# B&R Automation Studio project DuctLines (part 9)

### Program Logical/Uncoiler_1 (IEC)

#### Cyclic.ld
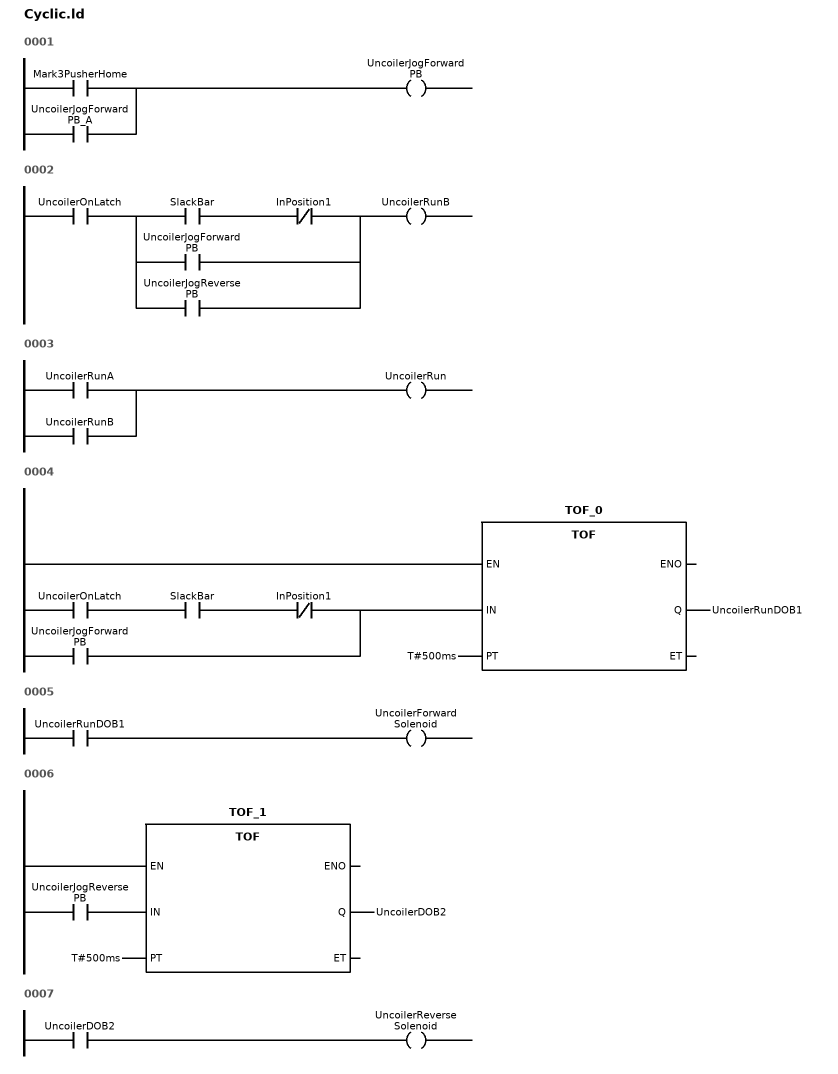
Ladder, written as Structured Text:
```iecst
PROGRAM _CYCLIC
(* Network 1 *)
UncoilerJogForwardPB := Mark3PusherHome OR UncoilerJogForwardPB_A;

(* Network 2 *)
UncoilerRunB := UncoilerOnLatch AND ((SlackBar AND NOT InPosition1) OR UncoilerJogForwardPB OR UncoilerJogReversePB);

(* Network 3 *)
UncoilerRun := UncoilerRunA OR UncoilerRunB;

(* Network 4 *)
TOF_0(IN := (UncoilerOnLatch AND SlackBar AND NOT InPosition1) OR UncoilerJogForwardPB, PT := T#500ms);
UncoilerRunDOB1 := TOF_0.Q;

(* Network 5 *)
UncoilerForwardSolenoid := UncoilerRunDOB1;

(* Network 6 *)
TOF_1(IN := UncoilerJogReversePB, PT := T#500ms);
UncoilerDOB2 := TOF_1.Q;

(* Network 7 *)
UncoilerReverseSolenoid := UncoilerDOB2;
END_PROGRAM
```

### Program Logical/E2Feeder (IEC) - 3/11/19 Punchmaster logic was redundant. Deleted rungs 169-189.

#### Variables.var
```iecst
VAR
	AutoSignal : BOOL;
	BatchCancelUnlatch : BOOL;
	BeadRollFires : BOOL;
	BeadRollUsedUp : BOOL;
	Block_1 : BOOL;
	BrakeLatch : BOOL;
	ButtonBack7 : BOOL;
	ButtonFires : BOOL;
	ButtonUsedUp : BOOL;
	CenterHoleFires : BOOL;
	CenterHoleTime : TIME;
	CenterHoleUsedUp : BOOL;
	CenterPosA : BOOL;
	CenterShuttleIndex : INT;
	ChangeCShuttle : BOOL;
	ChangeJob1 : BOOL;
	ChangeRShuttle : BOOL;
	ClearEncoderSignal : BOOL;
	CleatFires : BOOL;
	CleatUsedUp : BOOL;
	CLPUnlatch : BOOL;
	CoilPowerTripPulse : BOOL;
	CShuttleUnlatch : BOOL;
	CustomLTFires : BOOL;
	CustomLTTime : TIME;
	CustomLTUsedUp : BOOL;
	CustomLTValve : BOOL;
	CustomVFires : BOOL;
	CustomVTime : TIME;
	CustomVUsedUp : BOOL;
	DamperLatch : BOOL;
	DamperResult : DINT;
	DataUpdated : BOOL;
	DDDoneTimer : TON;
	DieDelayDone : BOOL;
	DieUpTime : TIME;
	DirectionDelayDone : BOOL;
	DuctoAutoUnlatch : BOOL;
	FFCLatch : BOOL;
	FiveFootCoil : BOOL;
	FourFootCoil : BOOL;
	FourResult : DINT;
	GapPulse : BOOL;
	GapTP : BOOL;
	GTime : TIME;
	HalfUpdated1 : BOOL;
	HalfUpdated2 : BOOL;
	HolePunchSelecedtSolenoid : BOOL;
	IncPartsMade : BOOL;
	InitMoveSignal : BOOL;
	InPositionBand : REAL := 0.01;
	JobChanging : BOOL;
	JobsDifferent : BOOL;
	LeftHoleFires : BOOL;
	LeftHoleTime : TIME;
	LeftHoleUsedUp : BOOL;
	LeftPosA : BOOL;
	LTFires : BOOL;
	LTTime : TIME;
	LTUsedUp : BOOL;
	MarkAccumulator : REAL;
	MetalEncoderLatch : DINT;
	NewRunJobOk : BOOL;
	NextMoveComplete : BOOL;
	NextMoveLookAgain : BOOL;
	NoShearHits : BOOL;
	OGLatch : BOOL;
	OGResult : DINT;
	OneResult : DINT;
	OutsideLatch : BOOL;
	PartCutOff : BOOL;
	PartRefOK : BOOL;
	PunchCurrentSelect : DINT;
	ReturnCalculated : BOOL;
	ReturnComplete : BOOL;
	ReturnTarget : DINT;
	RightHoleFires : BOOL;
	RightHoleTime : TIME;
	RightHoleUsedUp : BOOL;
	RightPosA : BOOL;
	RollEnableUnlatch : BOOL;
	RShuttleUnlatch : BOOL;
	RTotalInches : REAL;
	RunSpeedCalculated : BOOL;
	SetConnectorChange : BOOL;
	ShearBrakeFires : BOOL;
	ShearBrakeUsedUp : BOOL;
	ShearFires : BOOL;
	ShearHitsLTZero : BOOL;
	shearTime : TIME;
	ShearUsedUp : BOOL;
	SHLT0 : BOOL;
	SixFootCoil : BOOL;
	SmallResult : REAL;
	Step04A : BOOL;
	Step05A : BOOL;
	Step05B : BOOL;
	Step06 : BOOL;
	Step07 : BOOL;
	Step08 : BOOL;
	Step09 : BOOL;
	Step10 : BOOL;
	Step15 : BOOL;
	Step16 : BOOL;
	Step17 : BOOL;
	Step18A : BOOL;
	Step20 : BOOL;
	Step22 : BOOL;
	ThirdOff1 : BOOL;
	ThirdOff2 : BOOL;
	ThirdOff3 : BOOL;
	TON_0 : TON;
	TON_1 : TON;
	TON_10 : TON;
	TON_Warning : TON;
	TP_0 : TP;
	TP_1 : TP;
	TP_2 : TP;
	TP_3 : TP;
	TP_4 : TP;
	TP_5 : TP;
	TP_6 : TP;
	TP_7 : TP;
	TP_8 : TP;
	TP_9 : TP;
	TP_10 : TP;
	UnlatchBender : BOOL;
	UnlatchButtons : BOOL;
	VFires : BOOL;
	VTime : TIME;
	VUsedUp : BOOL;
	Wait1Ready : BOOL;
	Wait2Ready : BOOL;
	Wait3Ready : BOOL;
	WaitCon1 : BOOL;
	WaitCon2 : BOOL;
	ZCOLT0 : BOOL;
	ZCReverseComplete : BOOL;
	ZCSCTimer : TON;
	ZCSettleComplete : BOOL;
	ZeroCropDifference : DINT;
	ZRCTon : TON;
	FinalScan : BOOL;
	ShearAndDieFires : BOOL;
	DieDoneTimer : BOOL;
	TP_11 : TP;
END_VAR
```

#### Action.st
```iecst
ACTION myAction:
	IF ShearHits < 120000 THEN
		ShearHits := ShearHits + 1;
	END_IF;

END_ACTION

ACTION getNextMove:
	(*Find smallest move*)
	(*The shear will always be used*)
	IF getNextMove.x AND NOT getNextMove._x THEN
		FinalScan := TRUE;
	ELSE
		NextMoveDone := TRUE;
		SmallResult := ShearMove;
		IF LTNotchMove < SmallResult AND LTNotchMove > InvalidDistREAL THEN
			SmallResult := LTNotchMove;
		END_IF;
		IF VNotchMove < SmallResult AND VNotchMove > InvalidDistREAL THEN
			SmallResult := VNotchMove;
		END_IF;
		IF LeftHoleMove < SmallResult AND LeftHoleMove > InvalidDistREAL THEN
			SmallResult := LeftHoleMove;
		END_IF;
		IF CenterHoleMove < SmallResult AND CenterHoleMove > InvalidDistREAL THEN
			SmallResult := CenterHoleMove;
		END_IF;
		IF RightHoleMove < SmallResult AND RightHoleMove > InvalidDistREAL THEN
			SmallResult := RightHoleMove;
		END_IF;
		IF ButtonMove < SmallResult AND ButtonMove > InvalidDistREAL THEN
			SmallResult := ButtonMove;
		END_IF;
		IF ShearBrakeMove < SmallResult AND ShearBrakeMove > InvalidDistREAL THEN
			SmallResult := ShearBrakeMove;
		END_IF;
		IF CustomLTMove < SmallResult AND CustomLTMove > InvalidDistREAL THEN
			SmallResult := CustomLTMove;
		END_IF;
		IF CleatMove < SmallResult AND CleatMove > InvalidDistREAL THEN
			SmallResult := CleatMove;
		END_IF;
		IF CustomVMove < SmallResult AND CustomVMove > InvalidDistREAL THEN
			SmallResult := CustomVMove;
		END_IF;
		(*IF BeadRollMove < SmallResult AND BeadRollMove > InvalidDistREAL THEN
			SmallResult := BeadRollMove;
		END_IF;*)

		ShearMove := ShearMove - SmallResult;
		IF LTNotchMove > InvalidDistREAL THEN
			LTNotchMove := LTNotchMove - SmallResult;
		END_IF;
		IF VNotchMove > InvalidDistREAL THEN
			VNotchMove := VNotchMove - SmallResult;
		END_IF;
		IF LeftHoleMove > InvalidDistREAL THEN
			LeftHoleMove := LeftHoleMove - SmallResult;
		END_IF;
		IF CenterHoleMove > InvalidDistREAL THEN
			CenterHoleMove := CenterHoleMove - SmallResult;
		END_IF;
		IF RightHoleMove > InvalidDistREAL THEN
			RightHoleMove := RightHoleMove - SmallResult;
		END_IF;
		IF ButtonMove > InvalidDistREAL THEN
			ButtonMove := ButtonMove - SmallResult;
		END_IF;
		IF ShearBrakeMove > InvalidDistREAL THEN
			ShearBrakeMove := ShearBrakeMove - SmallResult;
		END_IF;
		IF CustomLTMove > InvalidDistREAL THEN
			CustomLTMove := CustomLTMove - SmallResult;
		END_IF;
		IF CleatMove > InvalidDistREAL THEN
			CleatMove := CleatMove - SmallResult;
		END_IF;
		IF CustomVMove > InvalidDistREAL THEN
			CustomVMove := CustomVMove - SmallResult;
		END_IF;
		(*IF BeadRollMove > InvalidDistREAL THEN
			BeadRollMove := BeadRollMove - SmallResult;
		END_IF;*)
	END_IF;
END_ACTION

ACTION UpdateTables:
	IF UpdateTables.x AND NOT UpdateTables._x THEN
		FinalScan := TRUE;
	ELSE
		UpdateTablesDone := TRUE;
		IF ShearUsedUp AND ShearHits > 0 THEN
			ShearFires := TRUE;
			ShearHits := ShearHits - 1;
			(*Do this before the index changes *)
			IF (ShearIndex = 0 AND ShearFFlag = 1) OR
				(ShearIndex = 1 AND ShearTable[2] <= InvalidDistREAL) OR
				(ShearIndex = 2) THEN
				PartCutOff := TRUE;
			END_IF;
			ShearIndex := ShearIndex + 1;
			IF ShearTable[ShearIndex] <= InvalidDistREAL THEN
				ShearIndex := 1;
			END_IF;
			IF ShearHits <= 0 THEN
				MakeShearTable := TRUE;
				ShearIndex := 0;
			END_IF;
		END_IF;
		IF LTUsedUp THEN
			IF LTNotchHits > 0 THEN
				LTFires := TRUE;
				LTNotchHits := LTNotchHits - 1;
			END_IF;
			LTNotchIndex := LTNotchIndex + 1;
			IF LTNotchTable[LTNotchIndex] <= InvalidDistREAL THEN
				LTNotchIndex := 1;
			END_IF;
			SavedConnector := LatestConnector;
			IF LTNotchHits <= 0 THEN
				MakeLTTable := TRUE;
				LTNotchIndex := 0;
			END_IF;
		END_IF;
		IF VUsedUp THEN
			IF VNotchHits > 0 THEN
				VFires := TRUE;
				VNotchHits := VNotchHits - 1;
			END_IF;
			VNotchIndex := VNotchIndex + 1;
			IF VNotchTable[VNotchIndex] <= InvalidDistREAL THEN
				VNotchIndex := 1;
			END_IF;
			IF VNotchHits <= 0 THEN
				MakeVTable := TRUE;
				VNotchIndex := 0;
			END_IF;
		END_IF;
		IF LeftHoleUsedUp THEN
			IF LeftHoleHits > 0 THEN
				LeftHoleFires := TRUE;
				LeftHoleHits := LeftHoleHits - 1;
			END_IF;
			LeftHoleIndex := LeftHoleIndex + 1;
			IF LeftHoleTable[LeftHoleIndex] <= InvalidDistREAL THEN
				LeftHoleIndex := 1;
			END_IF;
			IF LeftHoleHits <= 0 THEN
				MakeLHoleTable := TRUE;
				LeftHoleIndex := 0;
			END_IF;
		END_IF;
		IF CenterHoleUsedUp THEN
			IF CenterHoleHits > 0 THEN
				CenterHoleFires := TRUE;
				CenterHoleHits := CenterHoleHits - 1;
			END_IF;
			CenterHoleIndex := CenterHoleIndex + 1;
			IF CenterHoleTable[CenterHoleIndex] <= InvalidDistREAL THEN
				CenterHoleIndex := 1;
			END_IF;
			IF CenterHoleHits <= 0 THEN
				MakeCHoleTable := TRUE;
				CenterHoleIndex := 0;
			END_IF;
		END_IF;
		IF RightHoleUsedUp THEN
			IF RightHoleHits > 0 THEN
				RightHoleFires := TRUE;
				RightHoleHits := RightHoleHits - 1;
			END_IF;
			RightHoleIndex := RightHoleIndex + 1;
			IF RightHoleTable[RightHoleIndex] <= InvalidDistREAL THEN
				RightHoleIndex := 1;
			END_IF;
			IF RightHoleHits <= 0 THEN
				MakeRHoleTable := TRUE;
				RightHoleIndex := 0;
			END_IF;
		END_IF
		IF ButtonUsedUp THEN
			IF ButtonHits > 0 THEN
				ButtonFires := TRUE;
				ButtonHits := ButtonHits - 1;
			END_IF;
			ButtonIndex := ButtonIndex + 1;
			IF ButtonTable[ButtonIndex] <= InvalidDistREAL THEN
				ButtonIndex := 1;
			END_IF;
			IF ButtonHits <= 0 THEN
				MakeButtonTable := TRUE;
				ButtonIndex := 0;
			END_IF;
		END_IF;
		IF ShearBrakeUsedUp THEN
			IF ShearBrakeHits > 0 THEN
				ShearBrakeFires := TRUE;
				ShearBrakeHits := ShearBrakeHits - 1;
			END_IF;
			ShearBrakeIndex := ShearBrakeIndex + 1;
			IF ShearBrakeTable[ShearBrakeIndex] <= InvalidDistREAL THEN
				ShearBrakeIndex := 1;
			END_IF;
			IF ShearBrakeHits <= 0 THEN
				MakeShearBrakeTable := TRUE;
				ShearBrakeIndex := 0;
			END_IF;
		END_IF;
		IF CustomLTUsedUp THEN
			IF CustomLTHits > 0 THEN
				CustomLTFires := TRUE;
				CustomLTHits := CustomLTHits - 1;
			END_IF;
			CustomLTIndex := CustomLTIndex + 1;
			IF CustomLTTable[CustomLTIndex] <= InvalidDistREAL THEN
				CustomLTIndex := 1;
			END_IF;
			IF CustomLTHits <= 0 THEN
				MakeCustomLTTable := TRUE;
				CustomLTIndex := 0;
			END_IF;
		END_IF;
		IF CleatUsedUp THEN
			IF CleatHits > 0 THEN
				CleatFires := TRUE;
				CleatHits := CleatHits - 1;
			END_IF;
			CleatIndex := CleatIndex + 1;
			IF CleatTable[CleatIndex] <= InvalidDistREAL THEN
				CleatIndex := 1;
			END_IF;
			IF CleatHits <= 0 THEN
				MakeCleatTable := TRUE;
				CleatIndex := 0;
			END_IF;
		END_IF;
		IF CustomVUsedUp THEN
			IF CustomVHits > 0 THEN
				CustomVFires := TRUE;
				CustomVHits := CustomVHits - 1;
			END_IF;
			CustomVIndex := CustomVIndex + 1;
			IF CustomVTable[CustomVIndex] <= InvalidDistREAL THEN
				CustomVIndex := 1;
			END_IF;
			IF CustomVHits <= 0 THEN
				MakeCustomVTable := TRUE;
				CustomVIndex := 0;
			END_IF;
		END_IF;
		(*IF BeadRollUsedUp THEN
			IF BeadRollHits > 0 THEN
				BeadRollFires := TRUE;
				BeadRollHits := BeadRollHits - 1;
			END_IF;
			BeadRollIndex := BeadRollIndex + 1;
			IF BeadRollTable[BeadRollIndex] <= InvalidDistREAL THEN
				BeadRollIndex := 1;
			END_IF;
			IF BeadRollHits <= 0 THEN
				MakeBeadRollTable := TRUE;
				BeadRollIndex := 0;
			END_IF;
		END_IF; *)
	END_IF;
END_ACTION
```

#### Cyclic.ld
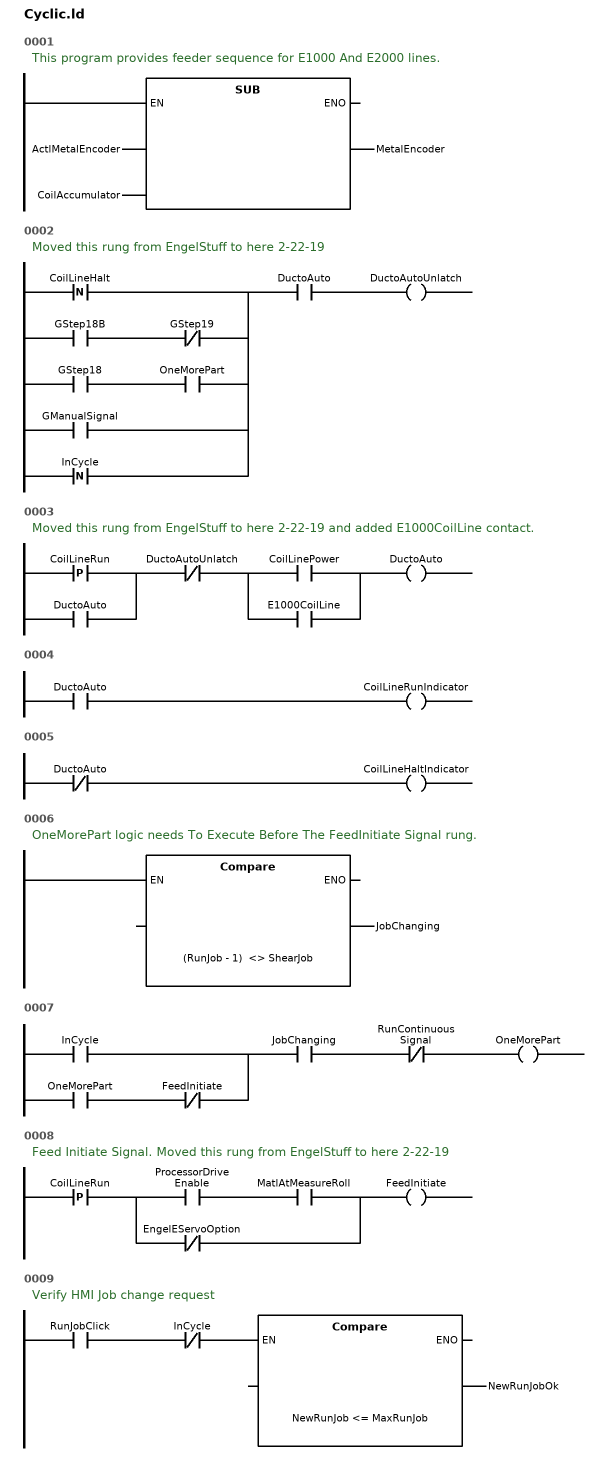
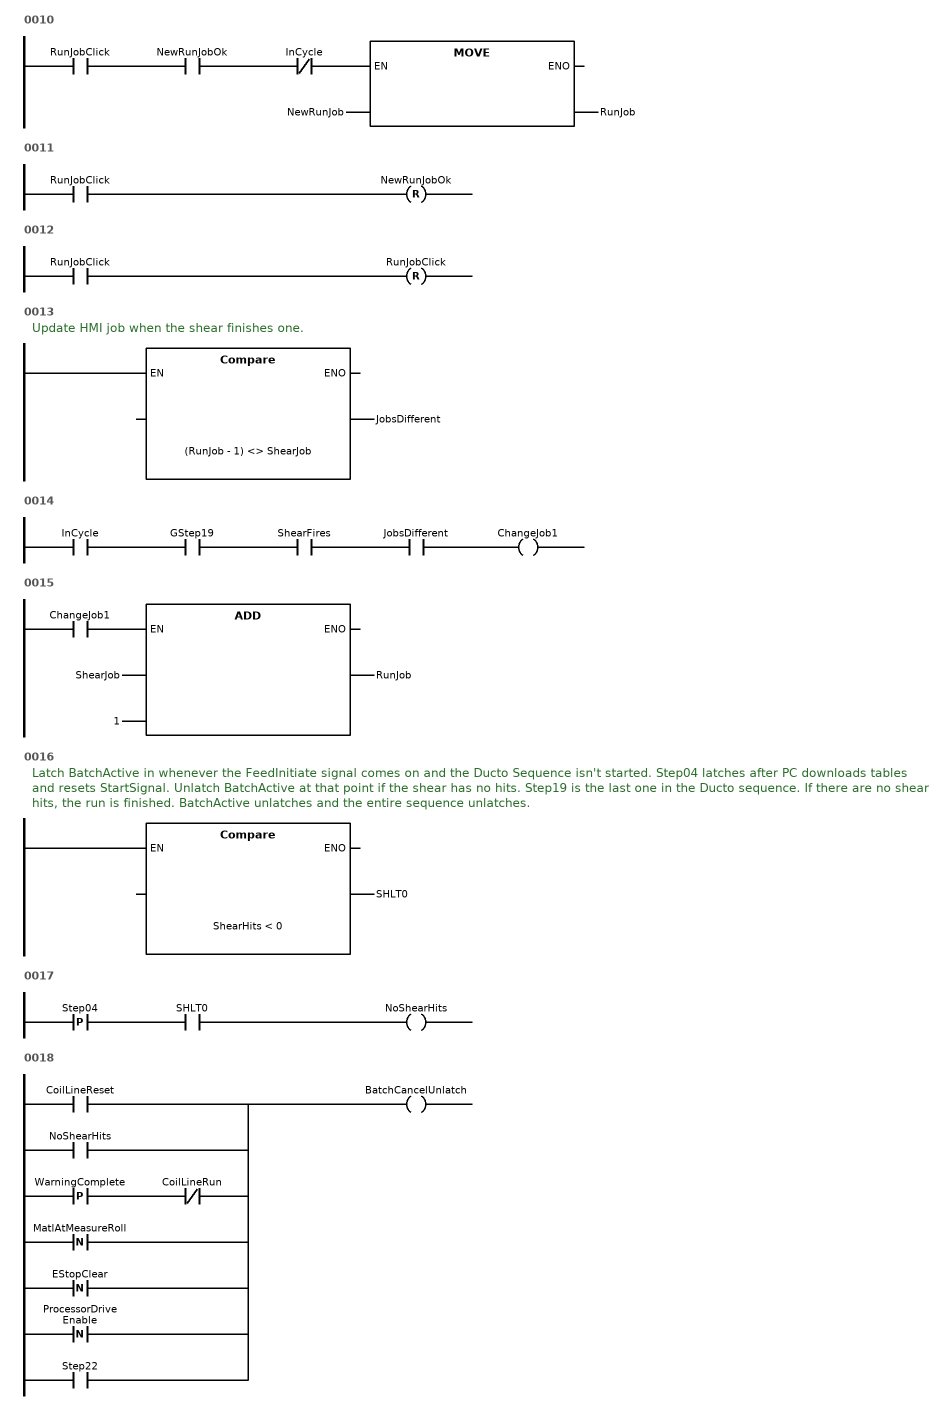
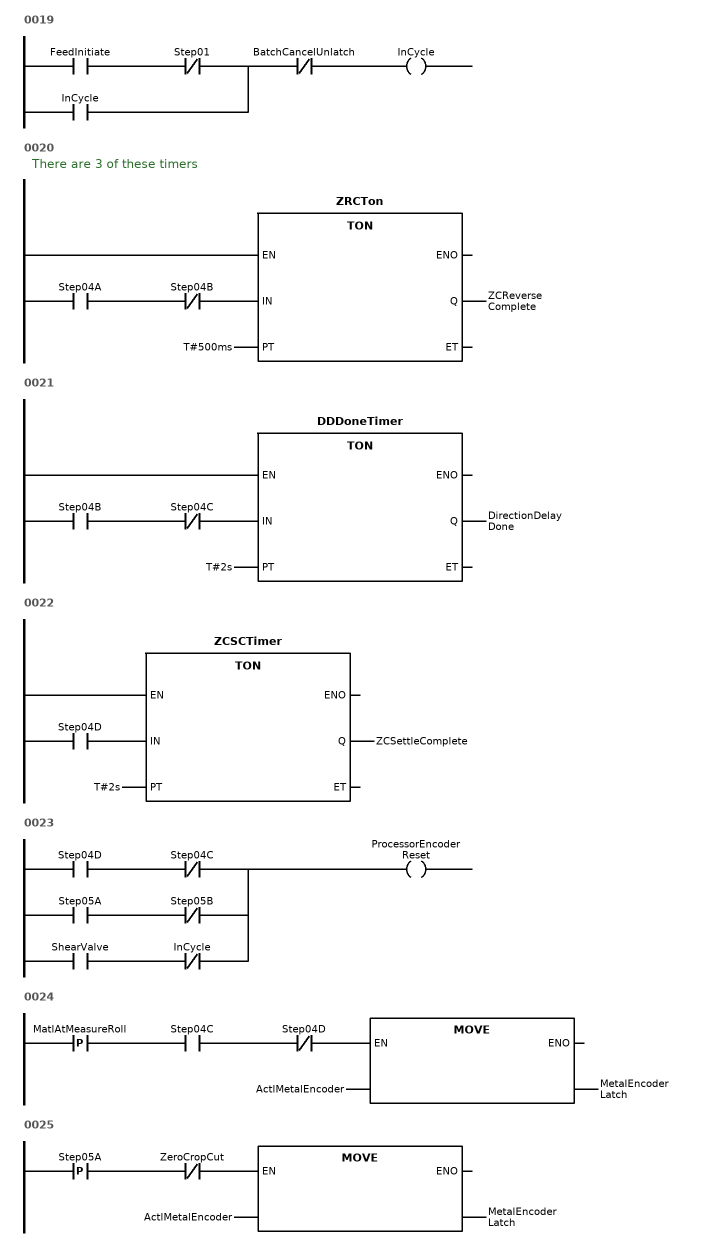
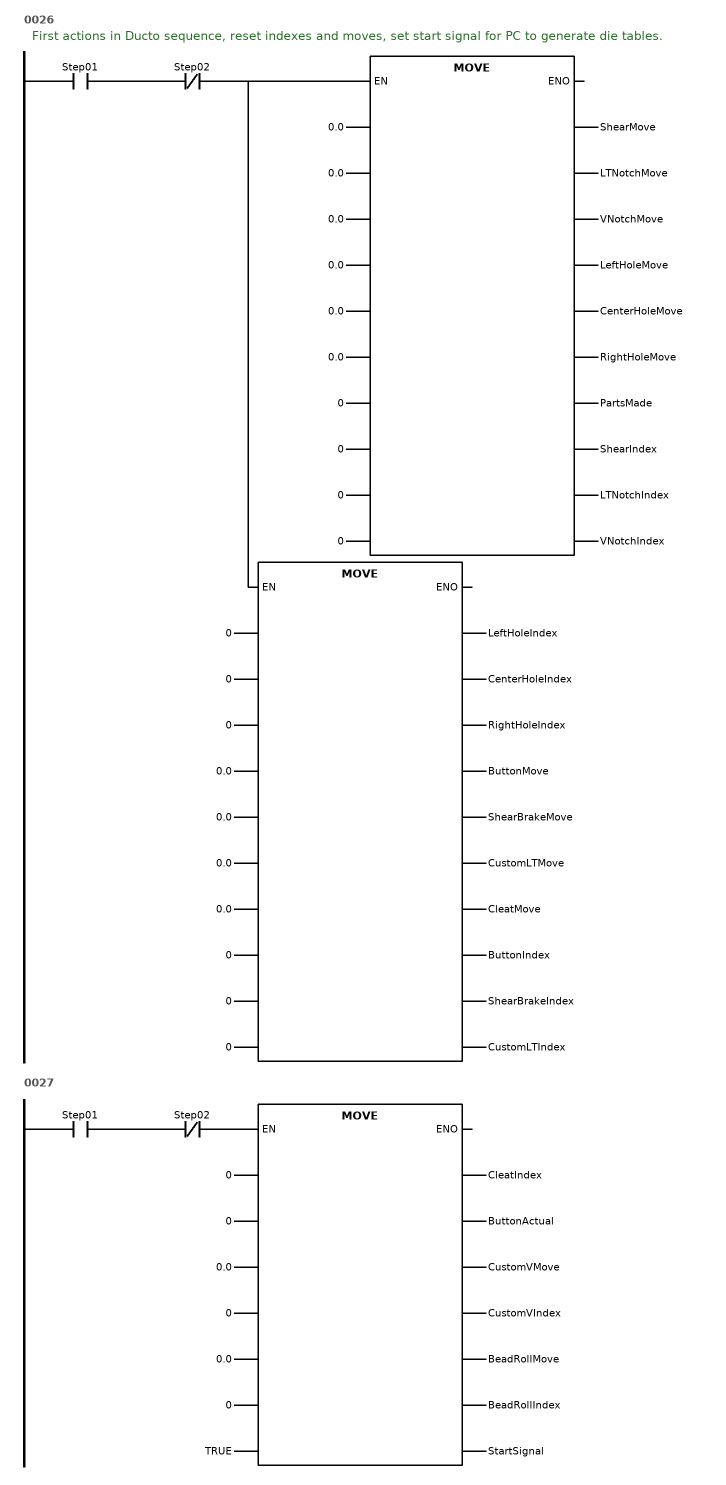
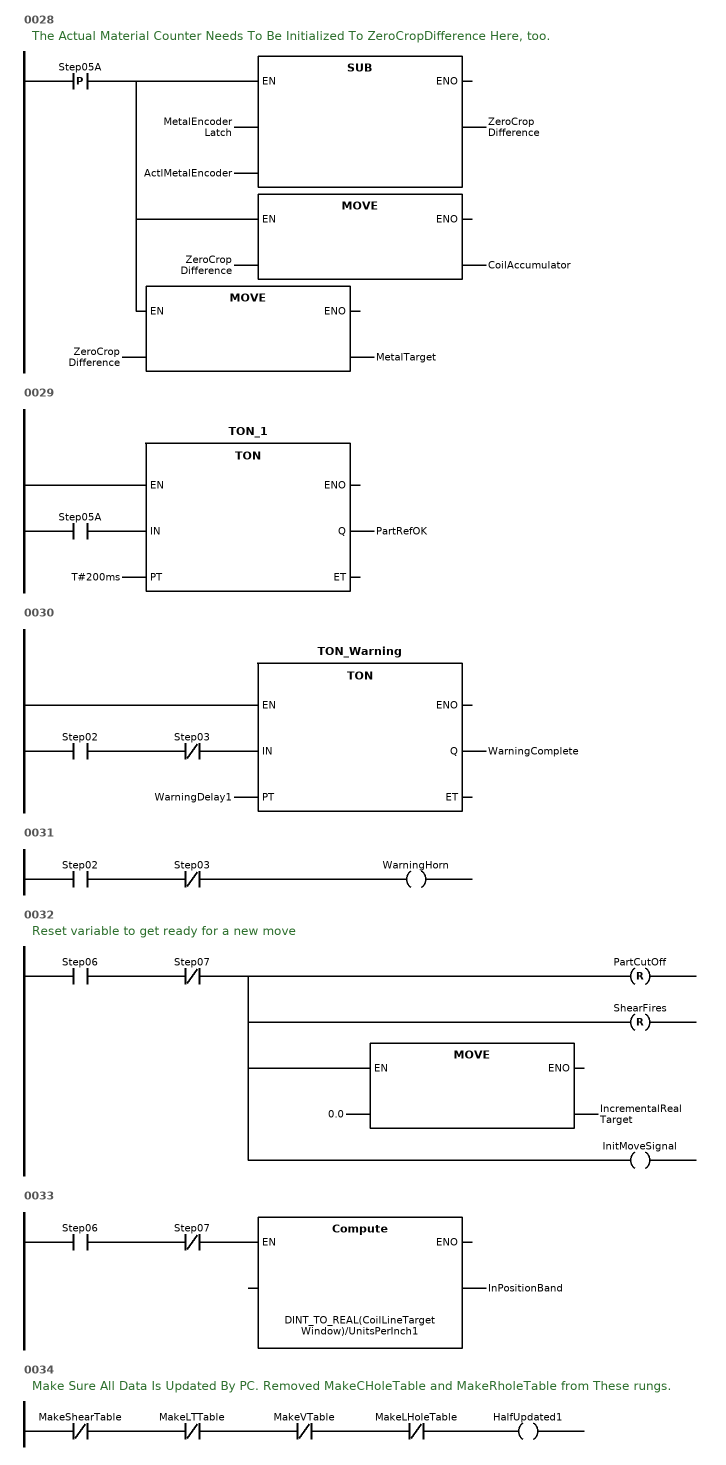
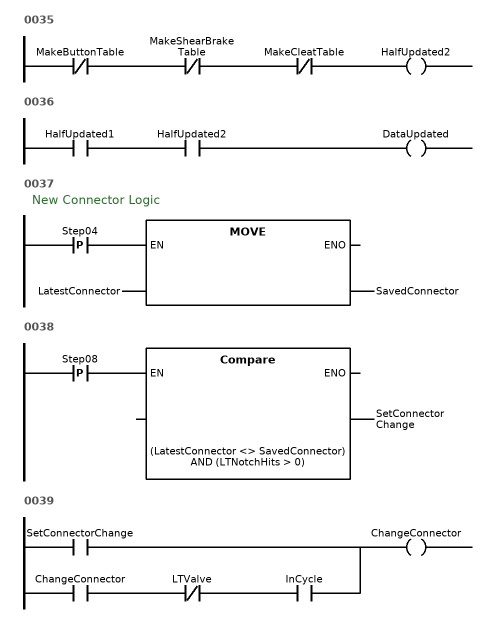
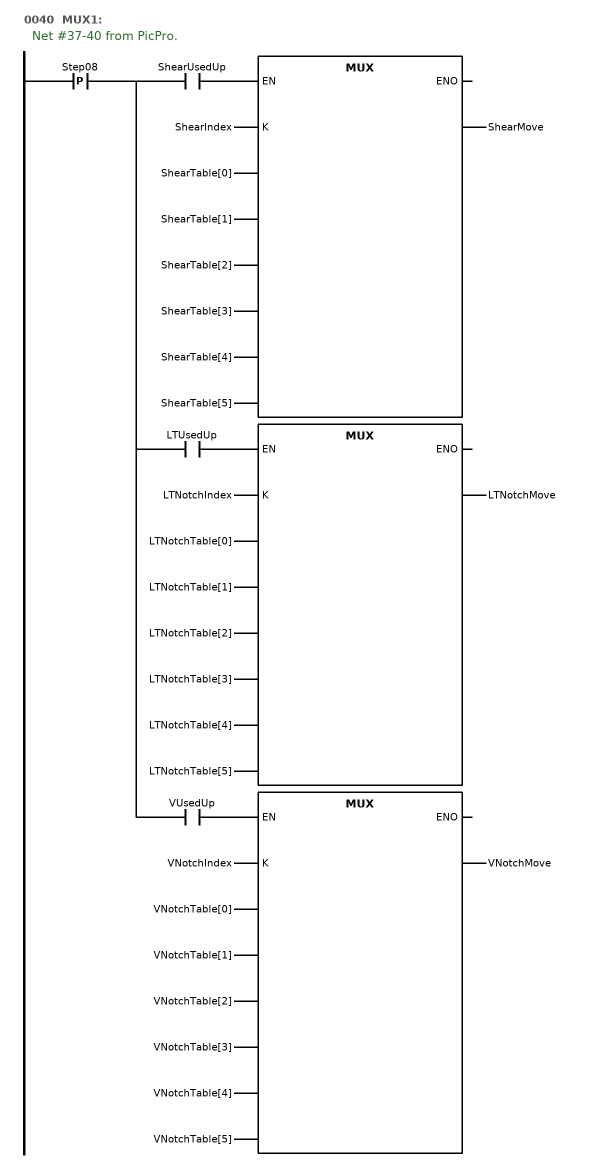
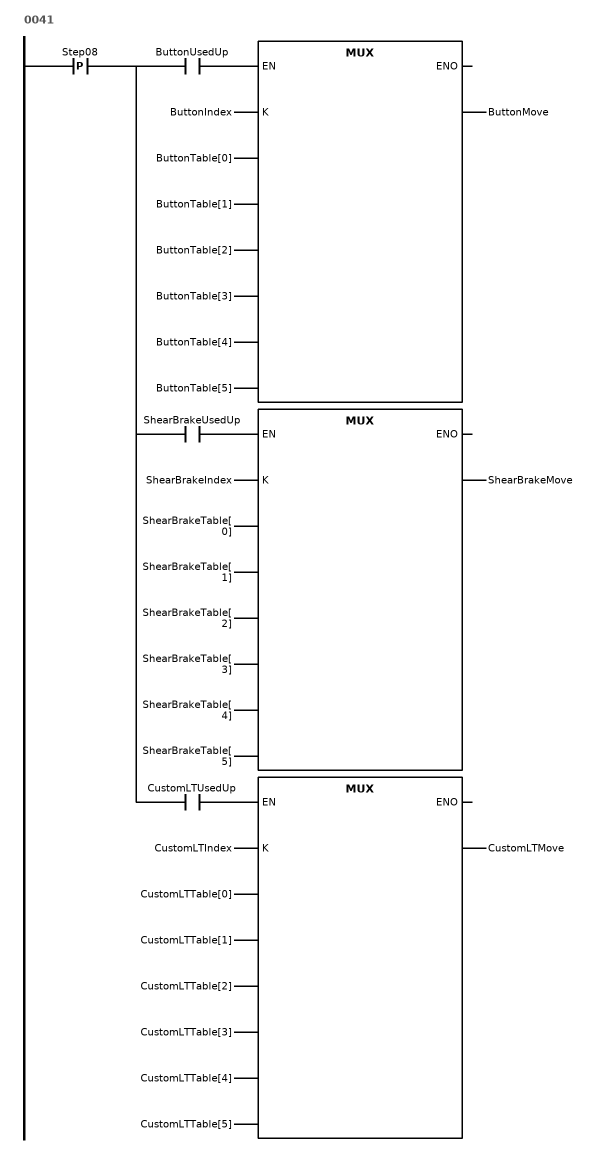
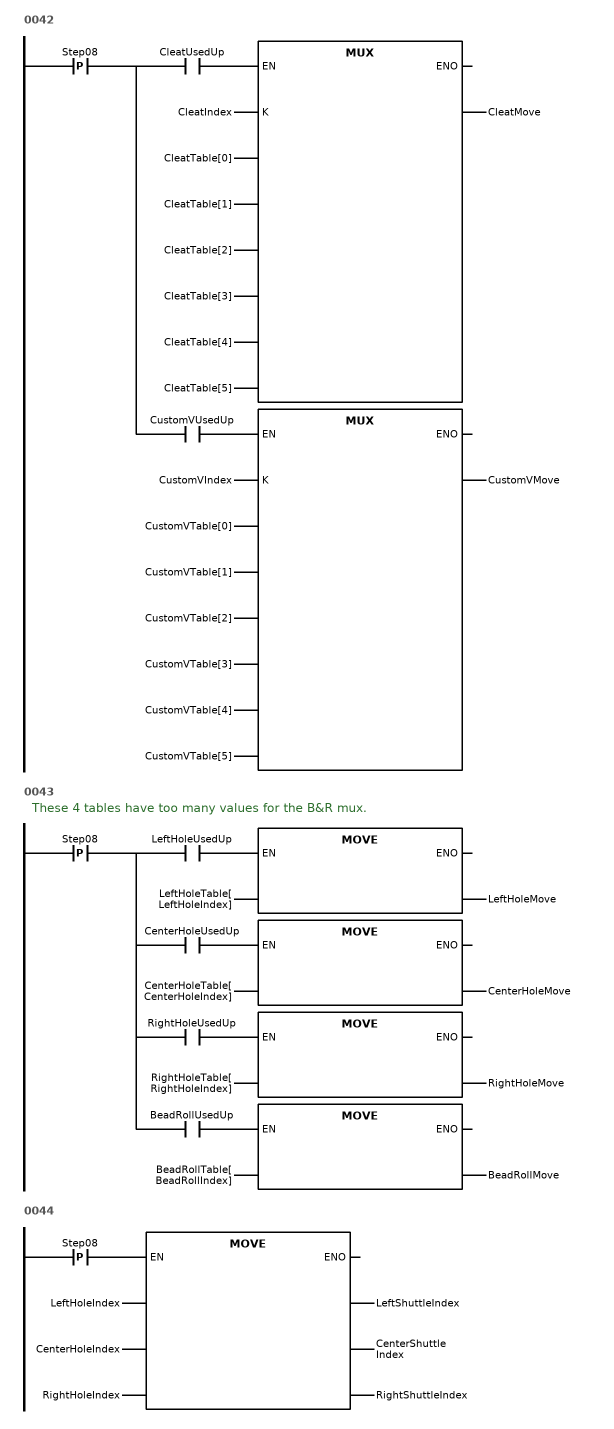
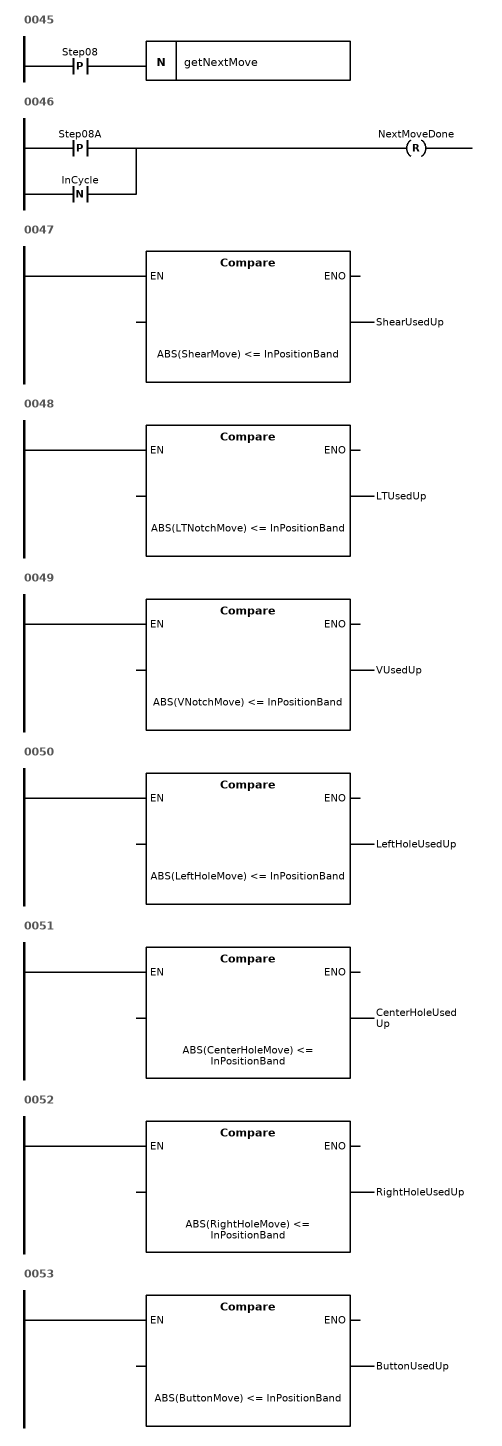
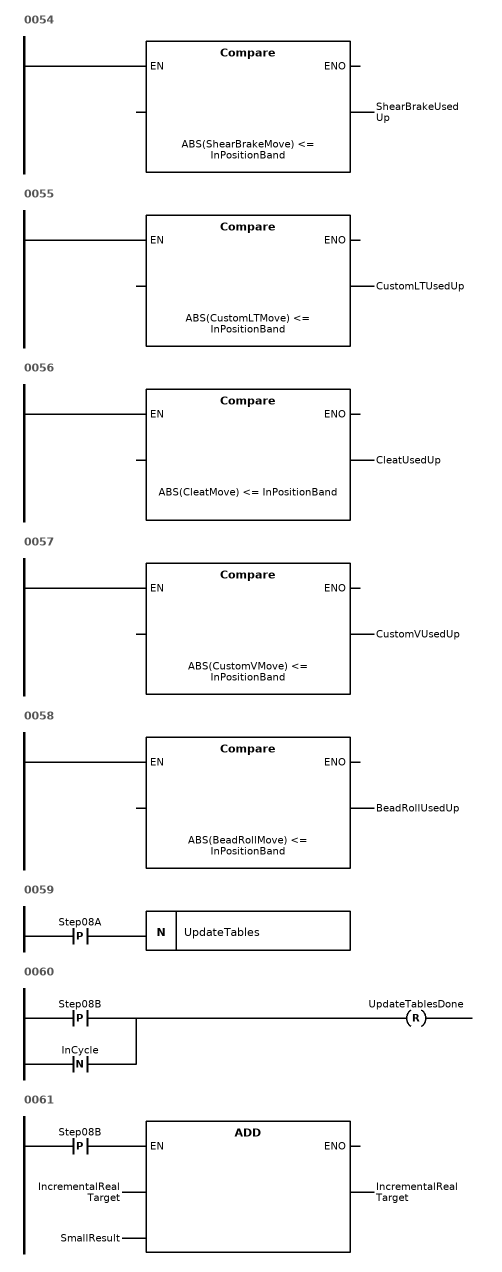
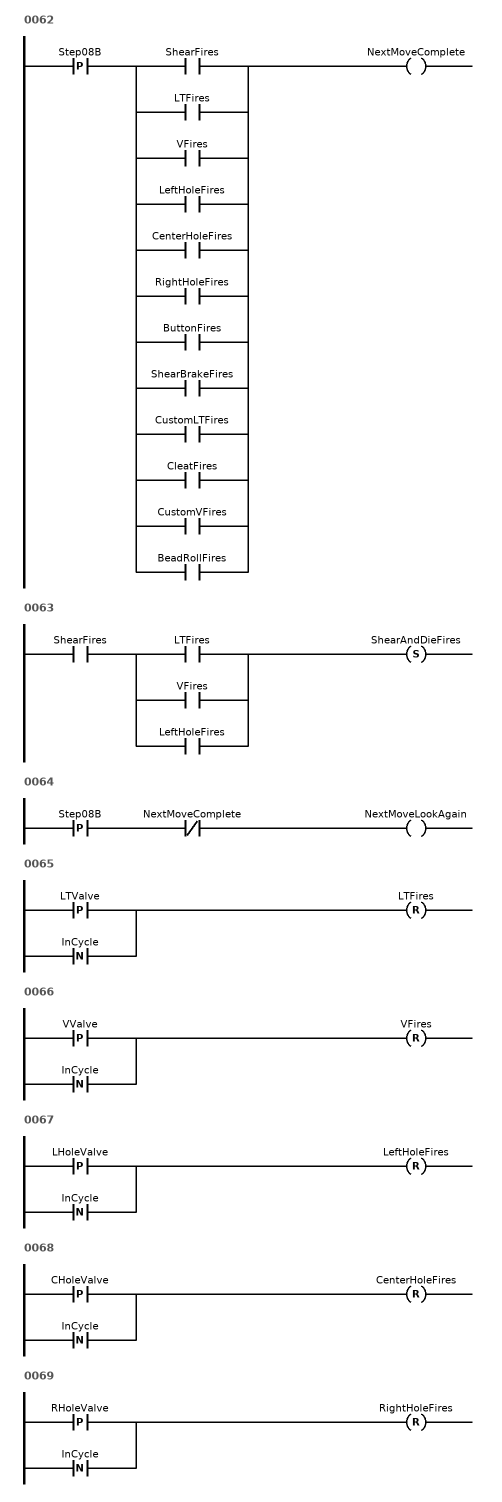
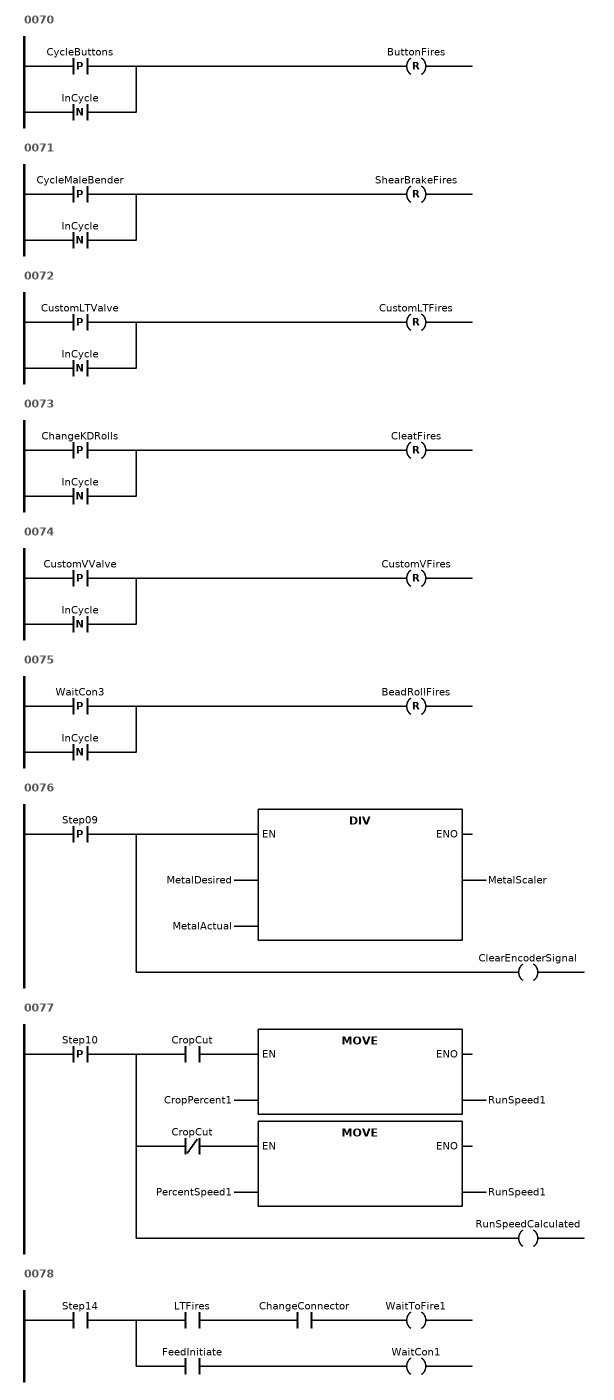
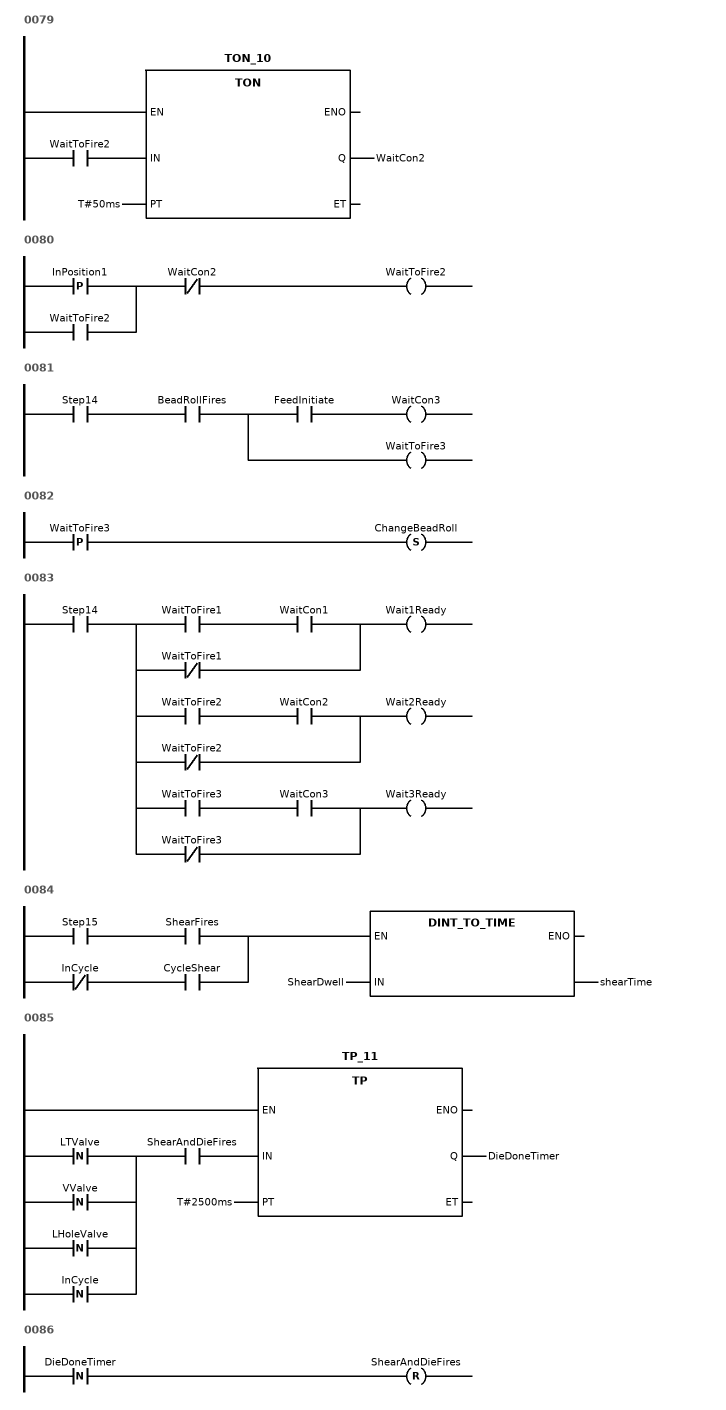
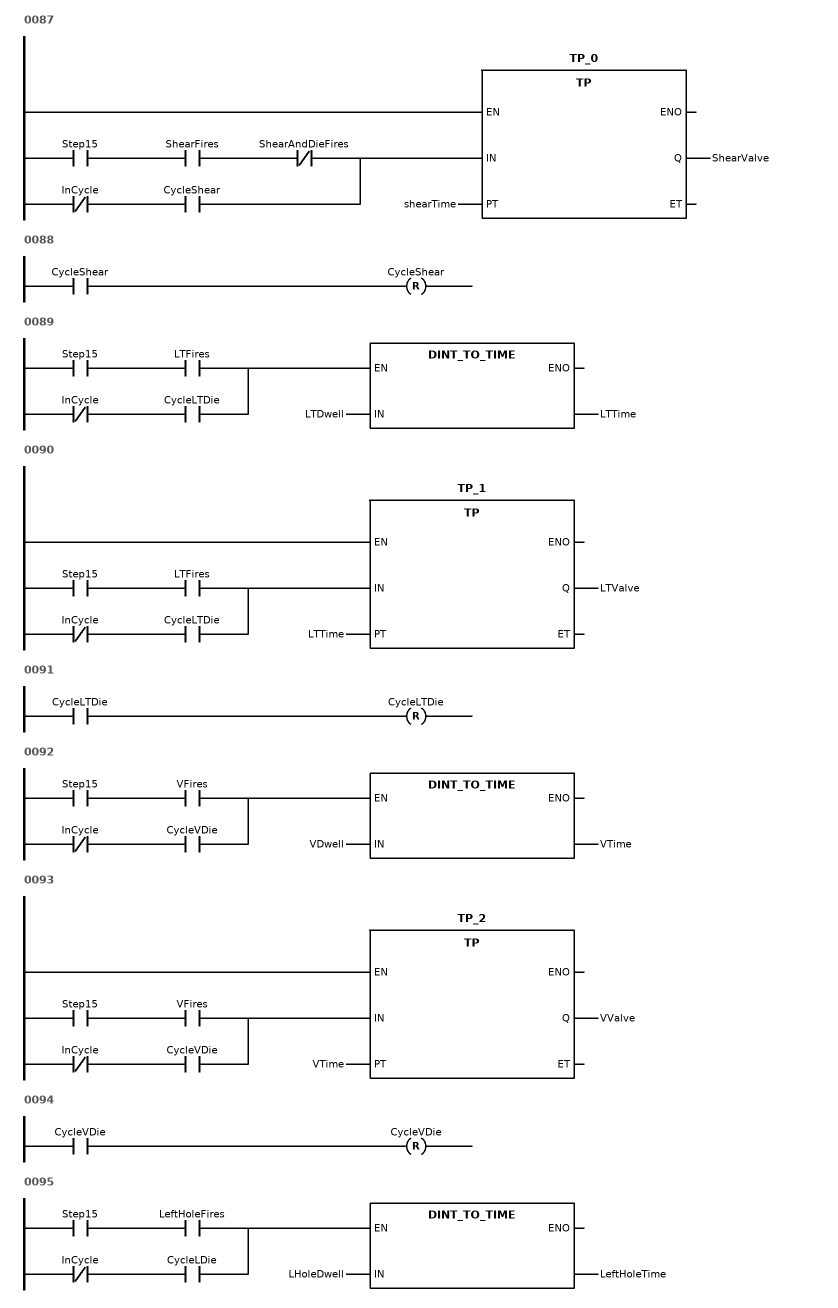
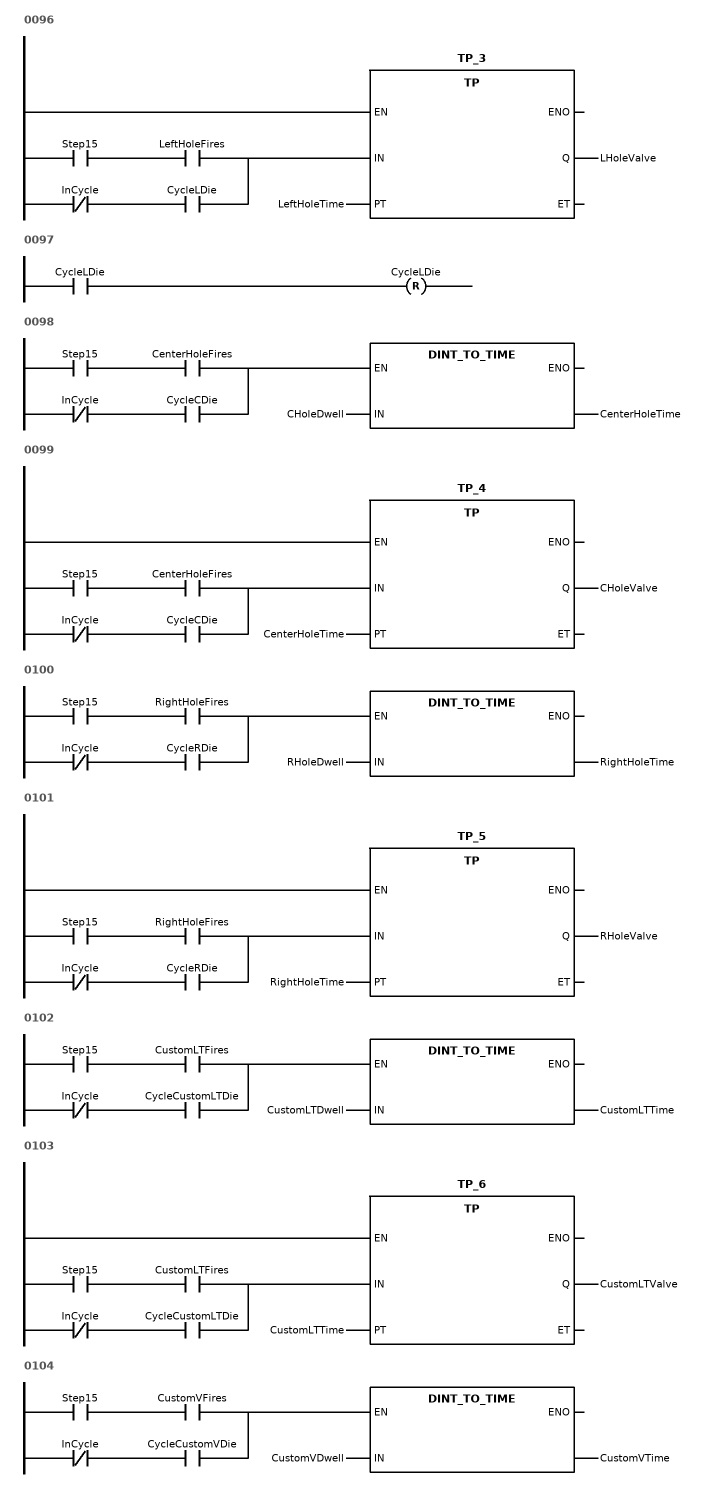
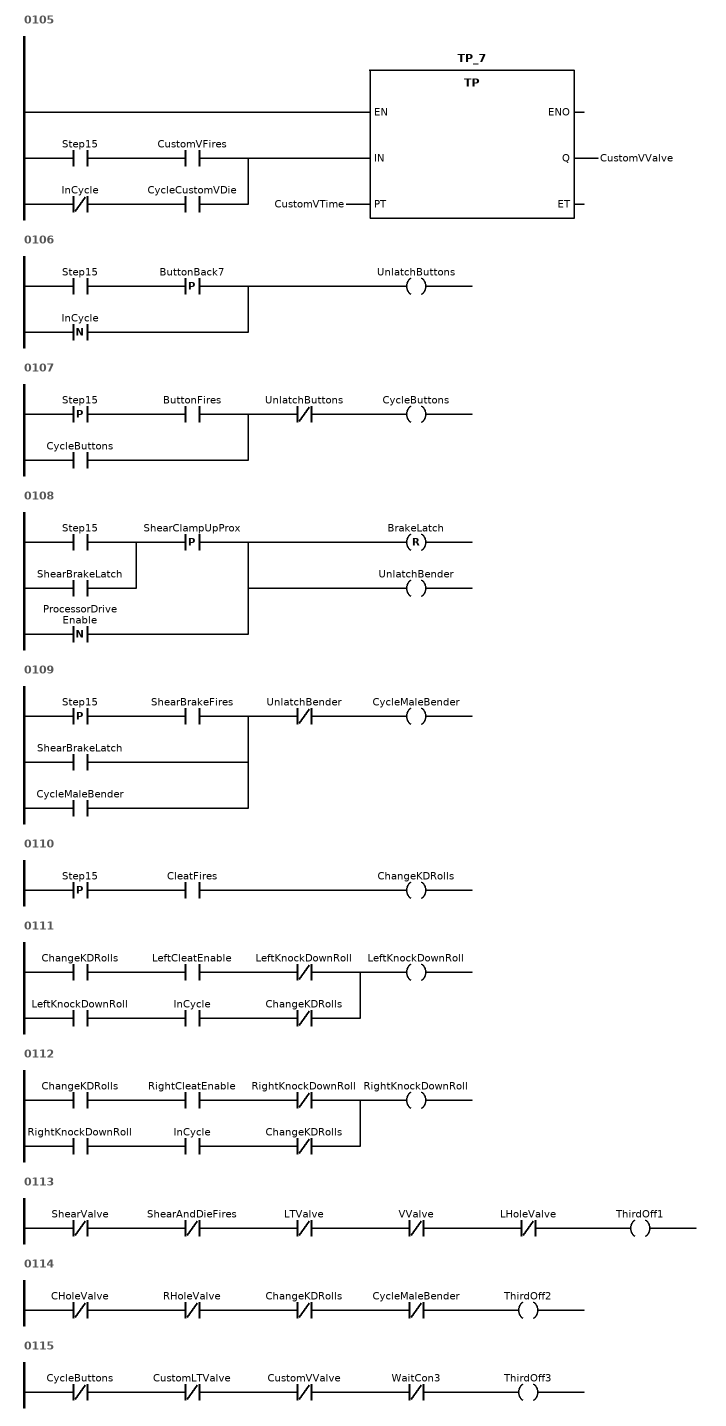
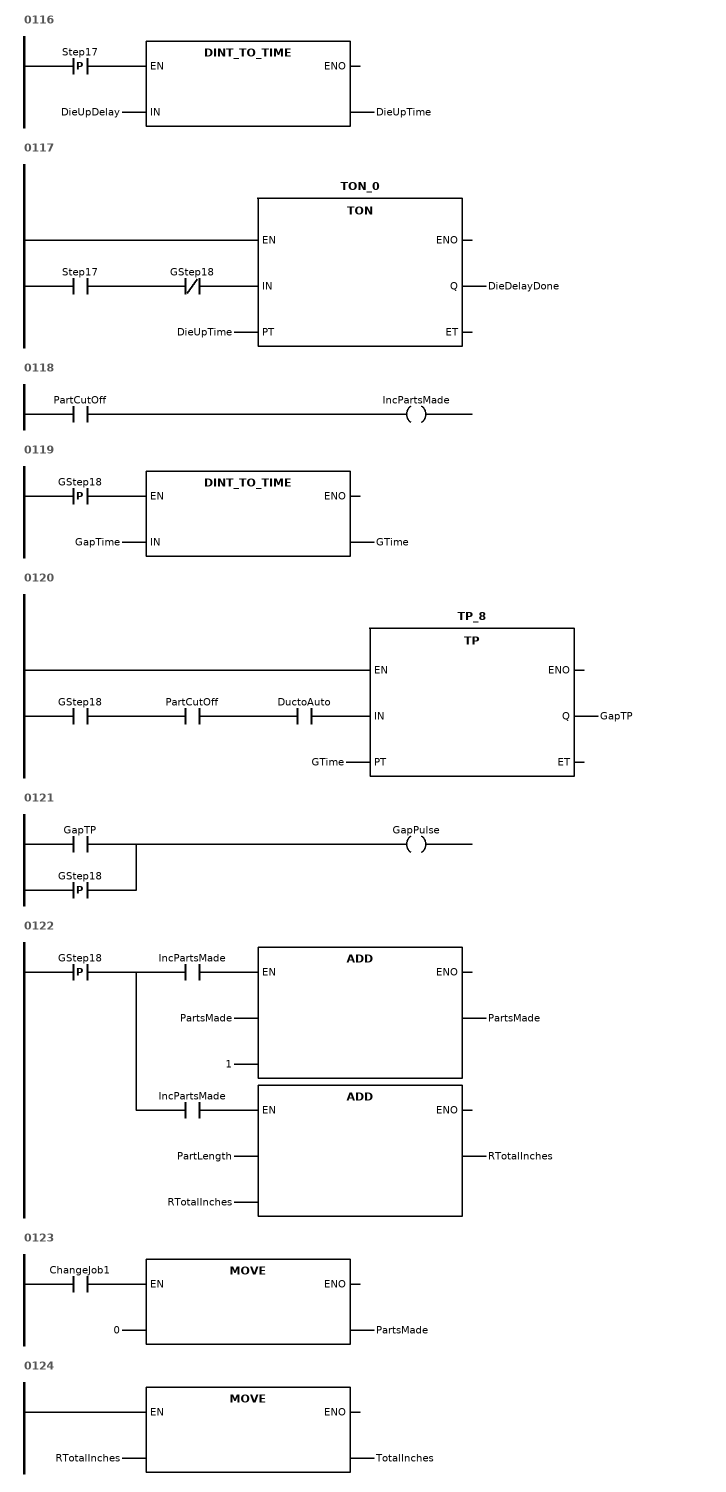
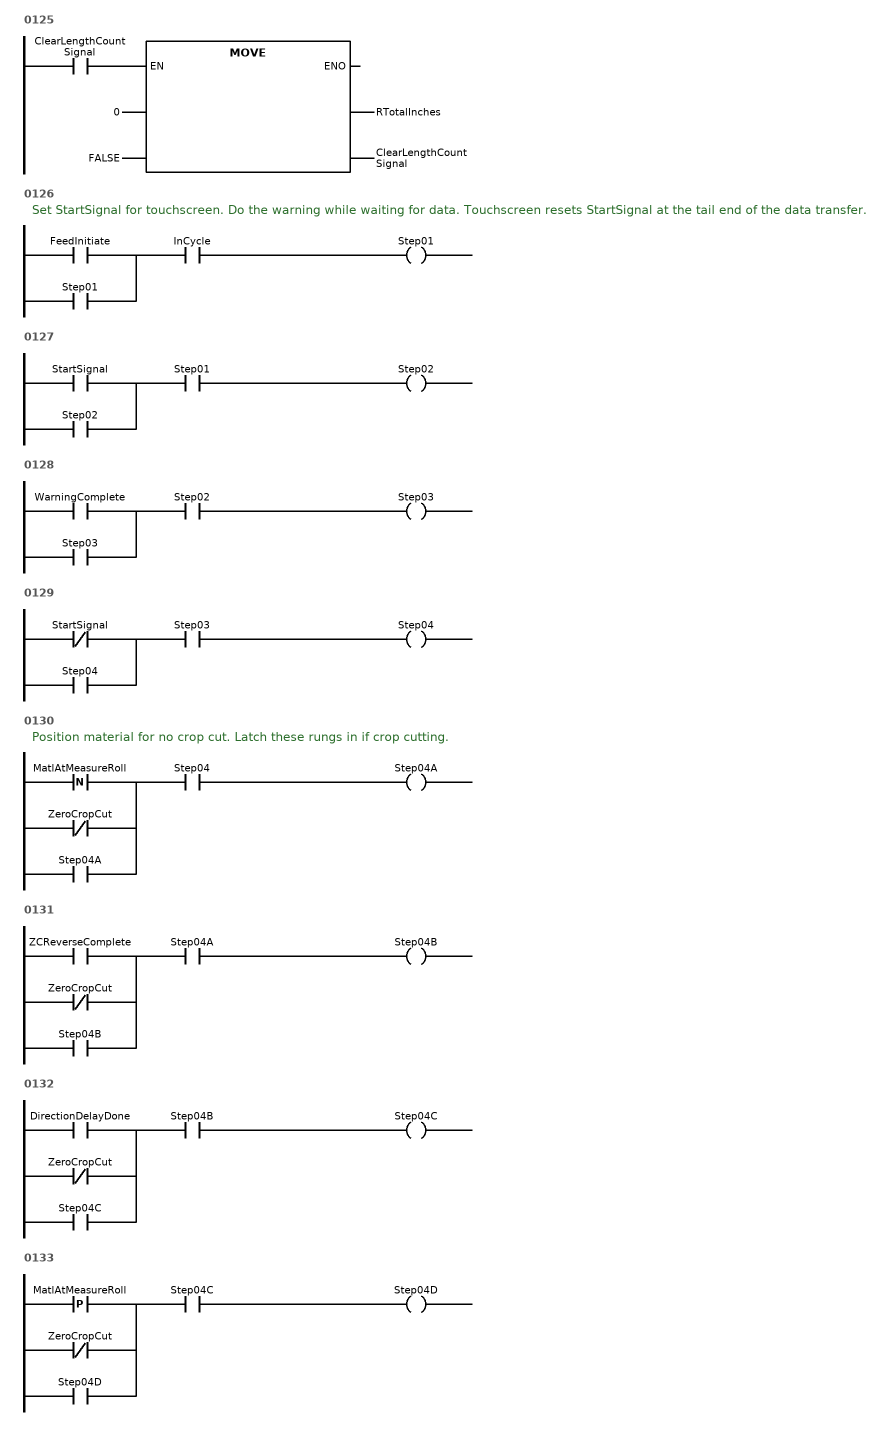
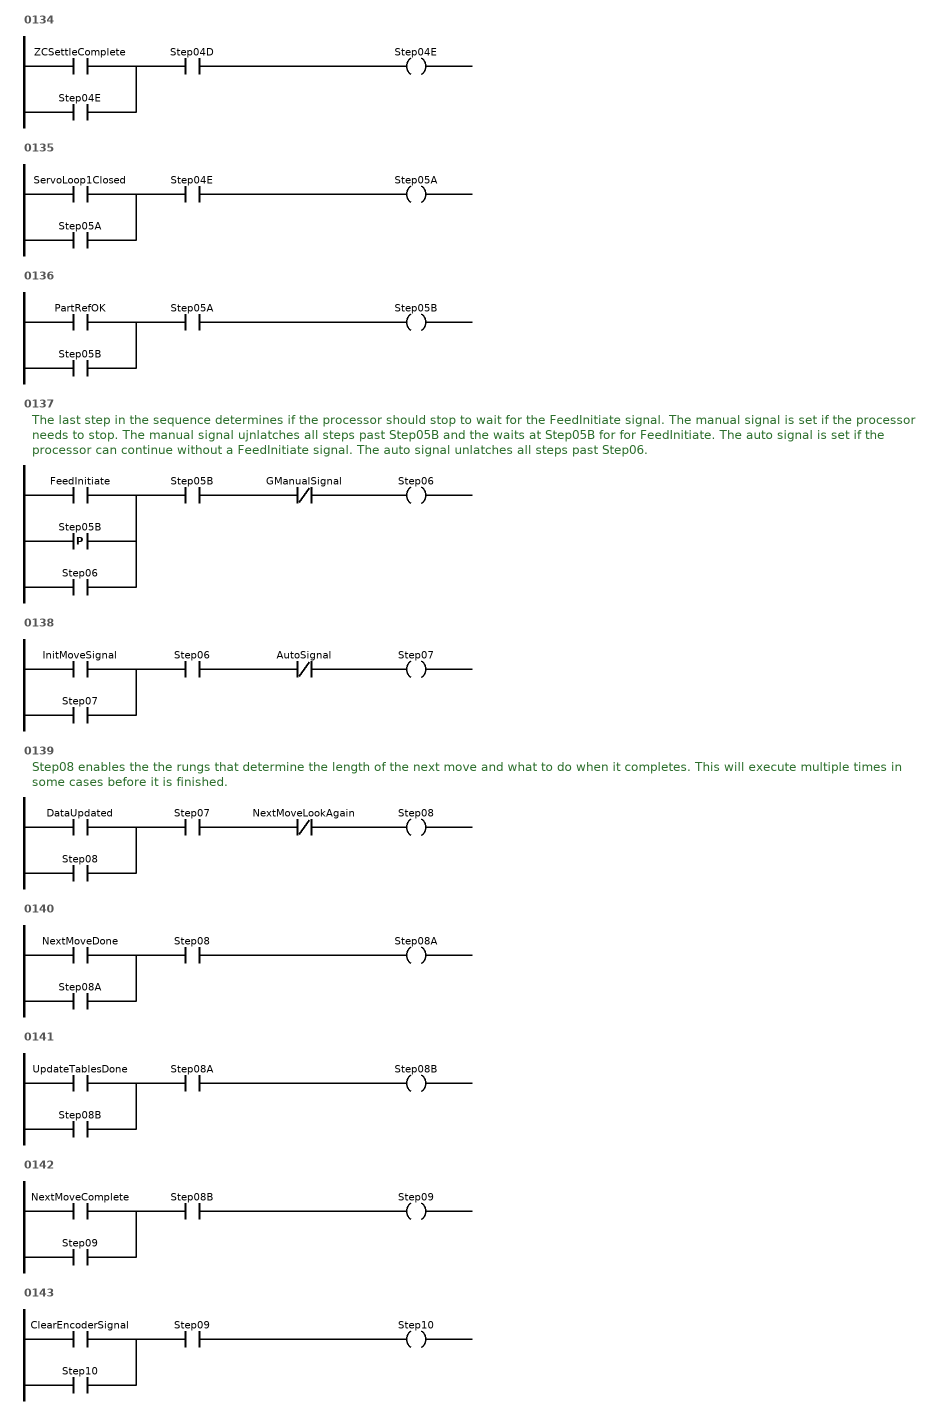
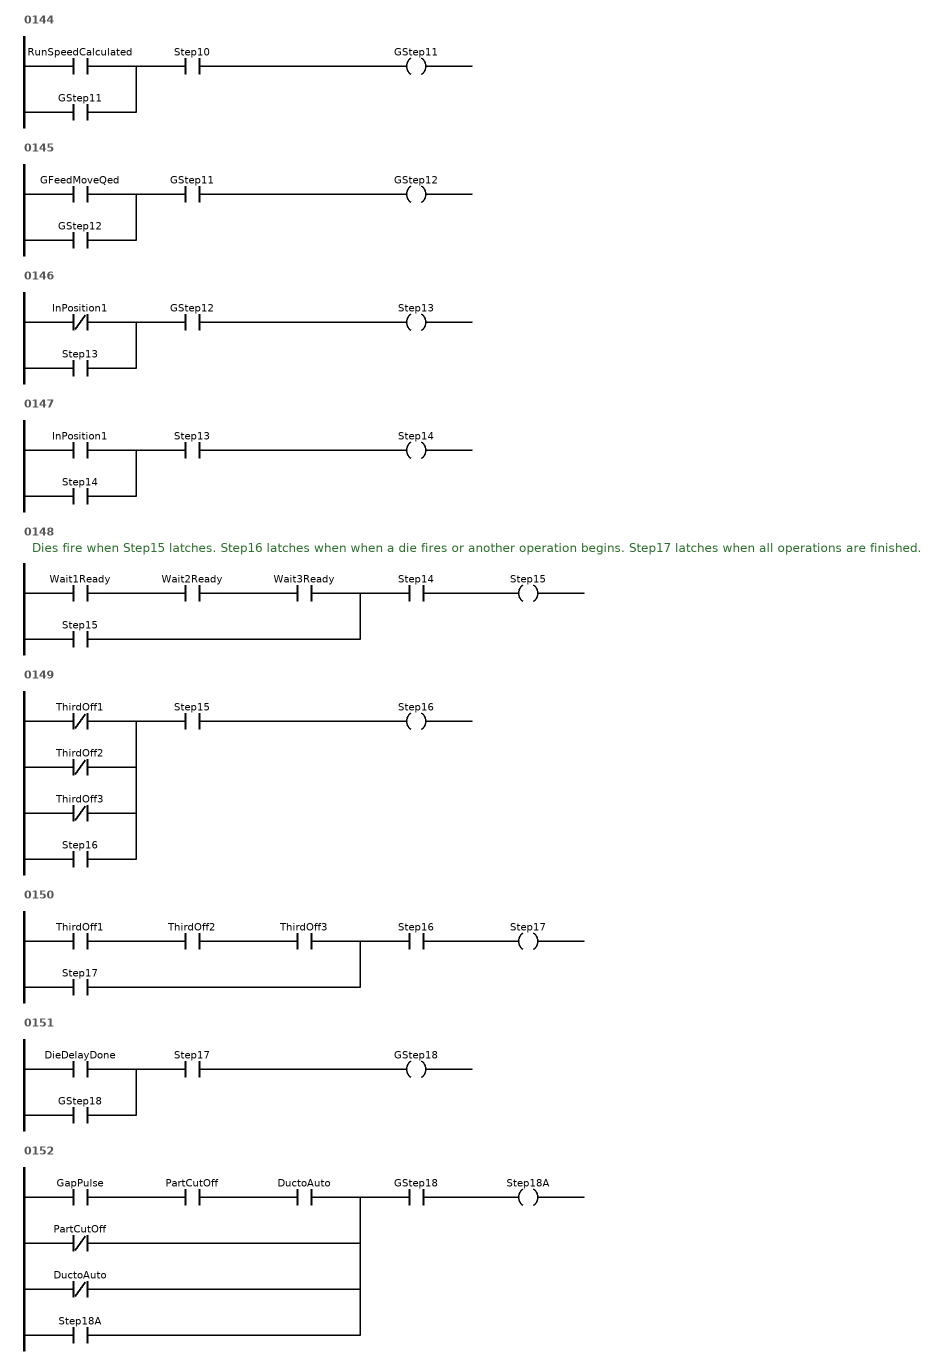
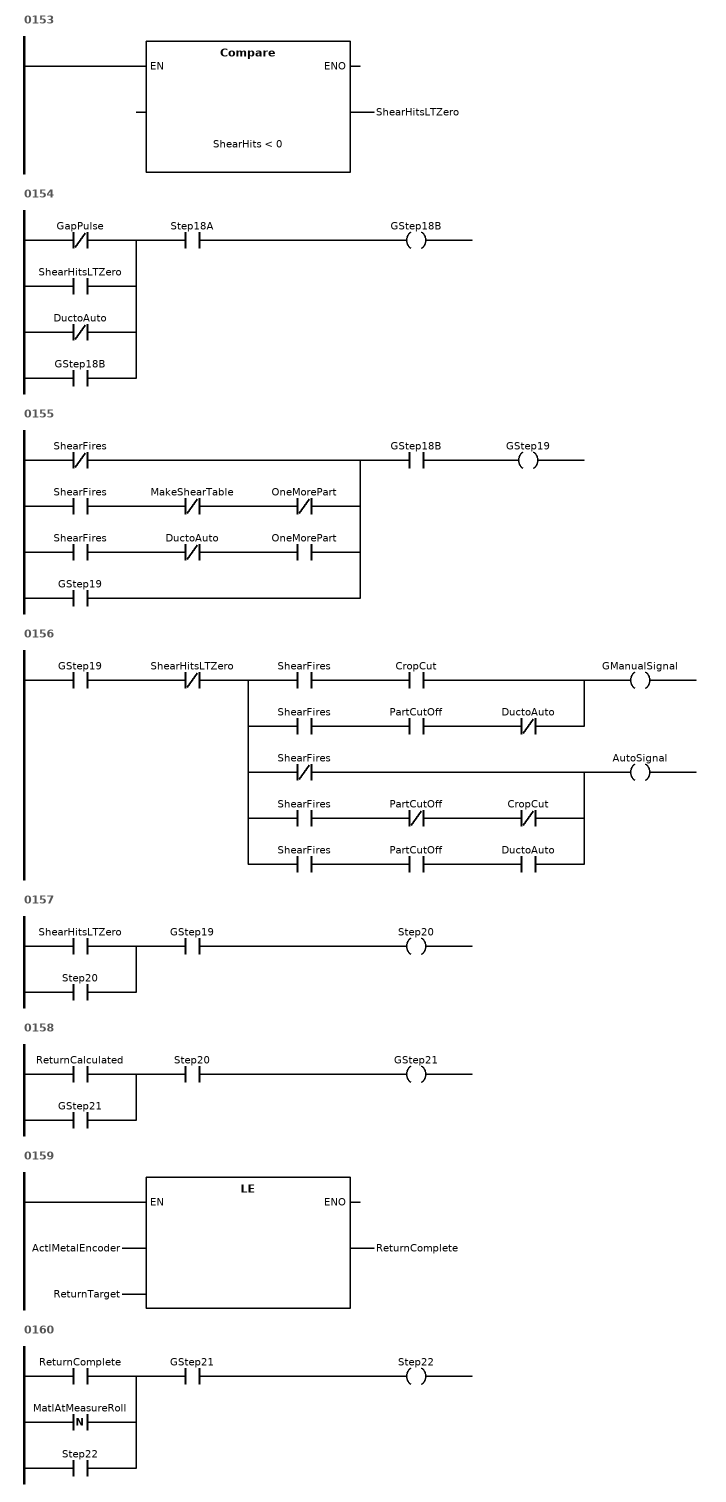
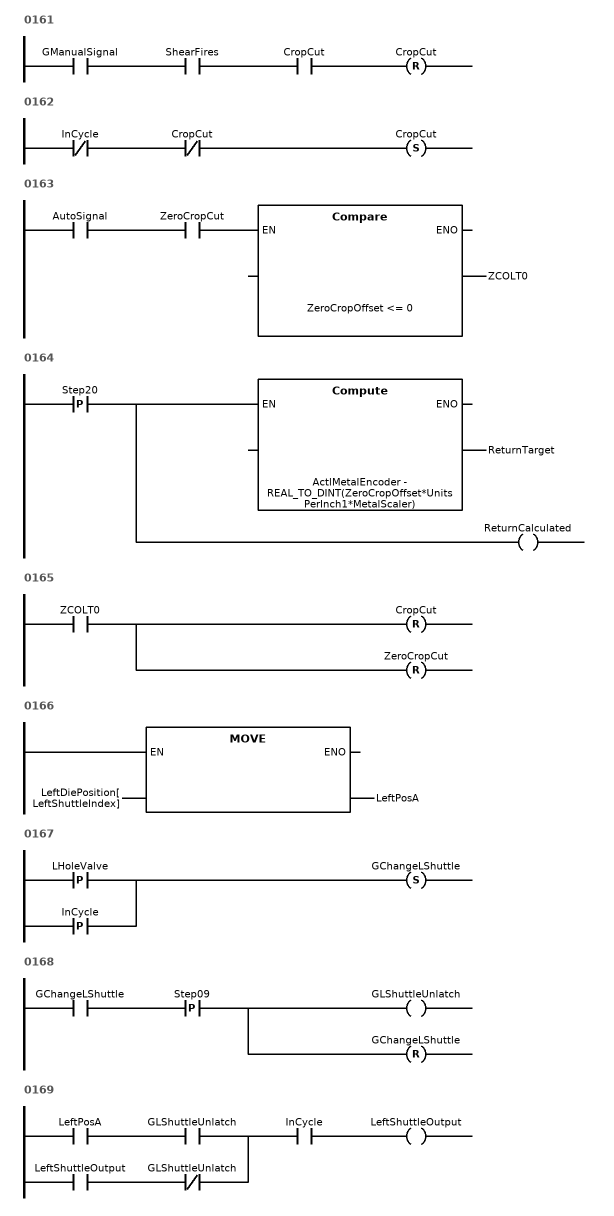
Ladder, written as Structured Text:
```iecst
PROGRAM _CYCLIC
VAR
    _e1 : F_TRIG;
    _e2 : F_TRIG;
    _e3 : R_TRIG;
    _e4 : R_TRIG;
    _e5 : R_TRIG;
    _e6 : R_TRIG;
    _e7 : F_TRIG;
    _e8 : F_TRIG;
    _e9 : F_TRIG;
    _e10 : R_TRIG;
    _e11 : R_TRIG;
    _e12 : R_TRIG;
    _e13 : R_TRIG;
    _e14 : R_TRIG;
    _e15 : R_TRIG;
    _e16 : R_TRIG;
    _e17 : R_TRIG;
    _e18 : R_TRIG;
    _e19 : R_TRIG;
    _e20 : R_TRIG;
    _e21 : R_TRIG;
    _e22 : F_TRIG;
    _e23 : R_TRIG;
    _e24 : R_TRIG;
    _e25 : F_TRIG;
    _e26 : R_TRIG;
    _e27 : R_TRIG;
    _e28 : R_TRIG;
    _e29 : R_TRIG;
    _e30 : F_TRIG;
    _e31 : R_TRIG;
    _e32 : F_TRIG;
    _e33 : R_TRIG;
    _e34 : F_TRIG;
    _e35 : R_TRIG;
    _e36 : F_TRIG;
    _e37 : R_TRIG;
    _e38 : F_TRIG;
    _e39 : R_TRIG;
    _e40 : F_TRIG;
    _e41 : R_TRIG;
    _e42 : F_TRIG;
    _e43 : R_TRIG;
    _e44 : F_TRIG;
    _e45 : R_TRIG;
    _e46 : F_TRIG;
    _e47 : R_TRIG;
    _e48 : F_TRIG;
    _e49 : R_TRIG;
    _e50 : F_TRIG;
    _e51 : R_TRIG;
    _e52 : R_TRIG;
    _e53 : R_TRIG;
    _e54 : R_TRIG;
    _e55 : F_TRIG;
    _e56 : F_TRIG;
    _e57 : F_TRIG;
    _e58 : F_TRIG;
    _e59 : F_TRIG;
    _e60 : R_TRIG;
    _e61 : F_TRIG;
    _e62 : R_TRIG;
    _e63 : R_TRIG;
    _e64 : F_TRIG;
    _e65 : R_TRIG;
    _e66 : R_TRIG;
    _e67 : R_TRIG;
    _e68 : R_TRIG;
    _e69 : R_TRIG;
    _e70 : R_TRIG;
    _p71 : BOOL;
    _e72 : F_TRIG;
    _e73 : R_TRIG;
    _e74 : R_TRIG;
    _e75 : F_TRIG;
    _e76 : R_TRIG;
    _e77 : R_TRIG;
    _e78 : R_TRIG;
    _e79 : R_TRIG;
END_VAR
(* Network 1: This program provides feeder sequence for E1000 And E2000 lines. *)
MetalEncoder := ActlMetalEncoder - CoilAccumulator;

(* Network 2: Moved this rung from EngelStuff to here 2-22-19 *)
_e1(CLK := CoilLineHalt);
_e2(CLK := InCycle);
DuctoAutoUnlatch := (_e1.Q OR (GStep18B AND NOT GStep19) OR (GStep18 AND OneMorePart) OR GManualSignal OR _e2.Q) AND DuctoAuto;

(* Network 3: Moved this rung from EngelStuff to here 2-22-19 and added E1000CoilLine contact. *)
_e3(CLK := CoilLineRun);
DuctoAuto := (_e3.Q OR DuctoAuto) AND NOT DuctoAutoUnlatch AND (CoilLinePower OR E1000CoilLine);

(* Network 4 *)
CoilLineRunIndicator := DuctoAuto;

(* Network 5 *)
CoilLineHaltIndicator := NOT DuctoAuto;

(* Network 6: OneMorePart logic needs To Execute Before The FeedInitiate Signal rung. *)
JobChanging := (RunJob - 1)  <> ShearJob;

(* Network 7 *)
OneMorePart := (InCycle OR (OneMorePart AND NOT FeedInitiate)) AND JobChanging AND NOT RunContinuousSignal;

(* Network 8: Feed Initiate Signal. Moved this rung from EngelStuff to here 2-22-19 *)
_e4(CLK := CoilLineRun);
FeedInitiate := _e4.Q AND ((ProcessorDriveEnable AND MatlAtMeasureRoll) OR NOT EngelEServoOption);

(* Network 9: Verify HMI Job change request *)
IF RunJobClick AND NOT InCycle THEN NewRunJobOk := NewRunJob <= MaxRunJob; END_IF;

(* Network 10 *)
IF RunJobClick AND NewRunJobOk AND NOT InCycle THEN RunJob := NewRunJob; END_IF;

(* Network 11 *)
IF RunJobClick THEN NewRunJobOk := FALSE; END_IF;

(* Network 12 *)
IF RunJobClick THEN RunJobClick := FALSE; END_IF;

(* Network 13: Update HMI job when the shear finishes one. *)
JobsDifferent := (RunJob - 1) <> ShearJob;

(* Network 14 *)
ChangeJob1 := InCycle AND GStep19 AND ShearFires AND JobsDifferent;

(* Network 15 *)
IF ChangeJob1 THEN RunJob := ShearJob + 1; END_IF;

(* Network 16: Latch BatchActive in whenever the FeedInitiate signal comes on and the Ducto Sequence isn't started. Step04 latches after PC downloads tables and resets StartSignal. Unlatch BatchActive at that point if the shear has no hits. Step19 is the last one in the Ducto sequence. If there are no shear hits, the run is finished. BatchActive unlatches and the entire sequence unlatches. *)
SHLT0 := ShearHits < 0;

(* Network 17 *)
_e5(CLK := Step04);
NoShearHits := _e5.Q AND SHLT0;

(* Network 18 *)
_e6(CLK := WarningComplete);
_e7(CLK := MatlAtMeasureRoll);
_e8(CLK := EStopClear);
_e9(CLK := ProcessorDriveEnable);
BatchCancelUnlatch := CoilLineReset OR NoShearHits OR (_e6.Q AND NOT CoilLineRun) OR _e7.Q OR _e8.Q OR _e9.Q OR Step22;

(* Network 19 *)
InCycle := ((FeedInitiate AND NOT Step01) OR InCycle) AND NOT BatchCancelUnlatch;

(* Network 20: There are 3 of these timers *)
ZRCTon(IN := Step04A AND NOT Step04B, PT := T#500ms);
ZCReverseComplete := ZRCTon.Q;

(* Network 21 *)
DDDoneTimer(IN := Step04B AND NOT Step04C, PT := T#2s);
DirectionDelayDone := DDDoneTimer.Q;

(* Network 22 *)
ZCSCTimer(IN := Step04D, PT := T#2s);
ZCSettleComplete := ZCSCTimer.Q;

(* Network 23 *)
ProcessorEncoderReset := (Step04D AND NOT Step04C) OR (Step05A AND NOT Step05B) OR (ShearValve AND NOT InCycle);

(* Network 24 *)
_e10(CLK := MatlAtMeasureRoll);
IF _e10.Q AND Step04C AND NOT Step04D THEN MetalEncoderLatch := ActlMetalEncoder; END_IF;

(* Network 25 *)
_e11(CLK := Step05A);
IF _e11.Q AND NOT ZeroCropCut THEN MetalEncoderLatch := ActlMetalEncoder; END_IF;

(* Network 26: First actions in Ducto sequence, reset indexes and moves, set start signal for PC to generate die tables. *)
IF Step01 AND NOT Step02 THEN
    ShearMove := 0.0;
    LTNotchMove := 0.0;
    VNotchMove := 0.0;
    LeftHoleMove := 0.0;
    CenterHoleMove := 0.0;
    RightHoleMove := 0.0;
    PartsMade := 0;
    ShearIndex := 0;
    LTNotchIndex := 0;
    VNotchIndex := 0;
    LeftHoleIndex := 0;
    CenterHoleIndex := 0;
    RightHoleIndex := 0;
    ButtonMove := 0.0;
    ShearBrakeMove := 0.0;
    CustomLTMove := 0.0;
    CleatMove := 0.0;
    ButtonIndex := 0;
    ShearBrakeIndex := 0;
    CustomLTIndex := 0;
END_IF;

(* Network 27 *)
IF Step01 AND NOT Step02 THEN
    CleatIndex := 0;
    ButtonActual := 0;
    CustomVMove := 0.0;
    CustomVIndex := 0;
    BeadRollMove := 0.0;
    BeadRollIndex := 0;
    StartSignal := TRUE;
END_IF;

(* Network 28: The Actual Material Counter Needs To Be Initialized To ZeroCropDifference Here, too. *)
_e12(CLK := Step05A);
IF _e12.Q THEN
    ZeroCropDifference := MetalEncoderLatch - ActlMetalEncoder;
    CoilAccumulator := ZeroCropDifference;
    MetalTarget := ZeroCropDifference;
END_IF;

(* Network 29 *)
TON_1(IN := Step05A, PT := T#200ms);
PartRefOK := TON_1.Q;

(* Network 30 *)
TON_Warning(IN := Step02 AND NOT Step03, PT := WarningDelay1);
WarningComplete := TON_Warning.Q;

(* Network 31 *)
WarningHorn := Step02 AND NOT Step03;

(* Network 32: Reset variable to get ready for a new move *)
IF Step06 AND NOT Step07 THEN
    PartCutOff := FALSE;
    ShearFires := FALSE;
    IncrementalRealTarget := 0.0;
END_IF;
InitMoveSignal := Step06 AND NOT Step07;

(* Network 33 *)
IF Step06 AND NOT Step07 THEN InPositionBand := DINT_TO_REAL(CoilLineTargetWindow)/UnitsPerInch1; END_IF;

(* Network 34: Make Sure All Data Is Updated By PC. Removed MakeCHoleTable and MakeRholeTable from These rungs. *)
HalfUpdated1 := NOT MakeShearTable AND NOT MakeLTTable AND NOT MakeVTable AND NOT MakeLHoleTable;

(* Network 35 *)
HalfUpdated2 := NOT MakeButtonTable AND NOT MakeShearBrakeTable AND NOT MakeCleatTable;

(* Network 36 *)
DataUpdated := HalfUpdated1 AND HalfUpdated2;

(* Network 37: New Connector Logic *)
_e13(CLK := Step04);
IF _e13.Q THEN SavedConnector := LatestConnector; END_IF;

(* Network 38 *)
_e14(CLK := Step08);
IF _e14.Q THEN SetConnectorChange := (LatestConnector <> SavedConnector) AND (LTNotchHits > 0); END_IF;

(* Network 39 *)
ChangeConnector := SetConnectorChange OR (ChangeConnector AND NOT LTValve AND InCycle);

(* Network 40: Net #37-40 from PicPro.  *)
MUX1:
_e15(CLK := Step08);
IF _e15.Q AND ShearUsedUp THEN
    ShearMove := MUX(K := ShearIndex, IN2 := ShearTable[0], IN3 := ShearTable[1], IN4 := ShearTable[2], IN5 := ShearTable[3], IN6 := ShearTable[4], IN7 := ShearTable[5]);
END_IF;
IF _e15.Q AND LTUsedUp THEN
    LTNotchMove := MUX(K := LTNotchIndex, IN2 := LTNotchTable[0], IN3 := LTNotchTable[1], IN4 := LTNotchTable[2], IN5 := LTNotchTable[3], IN6 := LTNotchTable[4], IN7 := LTNotchTable[5]);
END_IF;
IF _e15.Q AND VUsedUp THEN
    VNotchMove := MUX(K := VNotchIndex, IN2 := VNotchTable[0], IN3 := VNotchTable[1], IN4 := VNotchTable[2], IN5 := VNotchTable[3], IN6 := VNotchTable[4], IN7 := VNotchTable[5]);
END_IF;

(* Network 41 *)
_e16(CLK := Step08);
IF _e16.Q AND ButtonUsedUp THEN
    ButtonMove := MUX(K := ButtonIndex, IN2 := ButtonTable[0], IN3 := ButtonTable[1], IN4 := ButtonTable[2], IN5 := ButtonTable[3], IN6 := ButtonTable[4], IN7 := ButtonTable[5]);
END_IF;
IF _e16.Q AND ShearBrakeUsedUp THEN
    ShearBrakeMove := MUX(K := ShearBrakeIndex, IN2 := ShearBrakeTable[0], IN3 := ShearBrakeTable[1], IN4 := ShearBrakeTable[2], IN5 := ShearBrakeTable[3], IN6 := ShearBrakeTable[4], IN7 := ShearBrakeTable[5]);
END_IF;
IF _e16.Q AND CustomLTUsedUp THEN
    CustomLTMove := MUX(K := CustomLTIndex, IN2 := CustomLTTable[0], IN3 := CustomLTTable[1], IN4 := CustomLTTable[2], IN5 := CustomLTTable[3], IN6 := CustomLTTable[4], IN7 := CustomLTTable[5]);
END_IF;

(* Network 42 *)
_e17(CLK := Step08);
IF _e17.Q AND CleatUsedUp THEN
    CleatMove := MUX(K := CleatIndex, IN2 := CleatTable[0], IN3 := CleatTable[1], IN4 := CleatTable[2], IN5 := CleatTable[3], IN6 := CleatTable[4], IN7 := CleatTable[5]);
END_IF;
IF _e17.Q AND CustomVUsedUp THEN
    CustomVMove := MUX(K := CustomVIndex, IN2 := CustomVTable[0], IN3 := CustomVTable[1], IN4 := CustomVTable[2], IN5 := CustomVTable[3], IN6 := CustomVTable[4], IN7 := CustomVTable[5]);
END_IF;

(* Network 43: These 4 tables have too many values for the B&R mux. *)
_e18(CLK := Step08);
IF _e18.Q AND LeftHoleUsedUp THEN LeftHoleMove := LeftHoleTable[LeftHoleIndex]; END_IF;
IF _e18.Q AND CenterHoleUsedUp THEN CenterHoleMove := CenterHoleTable[CenterHoleIndex]; END_IF;
IF _e18.Q AND RightHoleUsedUp THEN RightHoleMove := RightHoleTable[RightHoleIndex]; END_IF;
IF _e18.Q AND BeadRollUsedUp THEN BeadRollMove := BeadRollTable[BeadRollIndex]; END_IF;

(* Network 44 *)
_e19(CLK := Step08);
IF _e19.Q THEN
    LeftShuttleIndex := LeftHoleIndex;
    CenterShuttleIndex := CenterHoleIndex;
    RightShuttleIndex := RightHoleIndex;
END_IF;

(* Network 45 *)
_e20(CLK := Step08);
IF _e20.Q THEN getNextMove; END_IF;

(* Network 46 *)
_e21(CLK := Step08A);
_e22(CLK := InCycle);
IF _e21.Q OR _e22.Q THEN NextMoveDone := FALSE; END_IF;

(* Network 47 *)
ShearUsedUp := ABS(ShearMove) <= InPositionBand;

(* Network 48 *)
LTUsedUp := ABS(LTNotchMove) <= InPositionBand;

(* Network 49 *)
VUsedUp := ABS(VNotchMove) <= InPositionBand;

(* Network 50 *)
LeftHoleUsedUp := ABS(LeftHoleMove) <= InPositionBand;

(* Network 51 *)
CenterHoleUsedUp := ABS(CenterHoleMove) <= InPositionBand;

(* Network 52 *)
RightHoleUsedUp := ABS(RightHoleMove) <= InPositionBand;

(* Network 53 *)
ButtonUsedUp := ABS(ButtonMove) <= InPositionBand;

(* Network 54 *)
ShearBrakeUsedUp := ABS(ShearBrakeMove) <= InPositionBand;

(* Network 55 *)
CustomLTUsedUp := ABS(CustomLTMove) <= InPositionBand;

(* Network 56 *)
CleatUsedUp := ABS(CleatMove) <= InPositionBand;

(* Network 57 *)
CustomVUsedUp := ABS(CustomVMove) <= InPositionBand;

(* Network 58 *)
BeadRollUsedUp := ABS(BeadRollMove) <= InPositionBand;

(* Network 59 *)
_e23(CLK := Step08A);
IF _e23.Q THEN UpdateTables; END_IF;

(* Network 60 *)
_e24(CLK := Step08B);
_e25(CLK := InCycle);
IF _e24.Q OR _e25.Q THEN UpdateTablesDone := FALSE; END_IF;

(* Network 61 *)
_e26(CLK := Step08B);
IF _e26.Q THEN IncrementalRealTarget := IncrementalRealTarget + SmallResult; END_IF;

(* Network 62 *)
_e27(CLK := Step08B);
NextMoveComplete := _e27.Q AND (ShearFires OR LTFires OR VFires OR LeftHoleFires OR CenterHoleFires OR RightHoleFires OR ButtonFires OR ShearBrakeFires OR CustomLTFires OR CleatFires OR CustomVFires OR BeadRollFires);

(* Network 63 *)
IF ShearFires AND (LTFires OR VFires OR LeftHoleFires) THEN ShearAndDieFires := TRUE; END_IF;

(* Network 64 *)
_e28(CLK := Step08B);
NextMoveLookAgain := _e28.Q AND NOT NextMoveComplete;

(* Network 65 *)
_e29(CLK := LTValve);
_e30(CLK := InCycle);
IF _e29.Q OR _e30.Q THEN LTFires := FALSE; END_IF;

(* Network 66 *)
_e31(CLK := VValve);
_e32(CLK := InCycle);
IF _e31.Q OR _e32.Q THEN VFires := FALSE; END_IF;

(* Network 67 *)
_e33(CLK := LHoleValve);
_e34(CLK := InCycle);
IF _e33.Q OR _e34.Q THEN LeftHoleFires := FALSE; END_IF;

(* Network 68 *)
_e35(CLK := CHoleValve);
_e36(CLK := InCycle);
IF _e35.Q OR _e36.Q THEN CenterHoleFires := FALSE; END_IF;

(* Network 69 *)
_e37(CLK := RHoleValve);
_e38(CLK := InCycle);
IF _e37.Q OR _e38.Q THEN RightHoleFires := FALSE; END_IF;

(* Network 70 *)
_e39(CLK := CycleButtons);
_e40(CLK := InCycle);
IF _e39.Q OR _e40.Q THEN ButtonFires := FALSE; END_IF;

(* Network 71 *)
_e41(CLK := CycleMaleBender);
_e42(CLK := InCycle);
IF _e41.Q OR _e42.Q THEN ShearBrakeFires := FALSE; END_IF;

(* Network 72 *)
_e43(CLK := CustomLTValve);
_e44(CLK := InCycle);
IF _e43.Q OR _e44.Q THEN CustomLTFires := FALSE; END_IF;

(* Network 73 *)
_e45(CLK := ChangeKDRolls);
_e46(CLK := InCycle);
IF _e45.Q OR _e46.Q THEN CleatFires := FALSE; END_IF;

(* Network 74 *)
_e47(CLK := CustomVValve);
_e48(CLK := InCycle);
IF _e47.Q OR _e48.Q THEN CustomVFires := FALSE; END_IF;

(* Network 75 *)
_e49(CLK := WaitCon3);
_e50(CLK := InCycle);
IF _e49.Q OR _e50.Q THEN BeadRollFires := FALSE; END_IF;

(* Network 76 *)
_e51(CLK := Step09);
IF _e51.Q THEN MetalScaler := MetalDesired / MetalActual; END_IF;
ClearEncoderSignal := _e51.Q;

(* Network 77 *)
_e52(CLK := Step10);
IF _e52.Q AND CropCut THEN RunSpeed1 := CropPercent1; END_IF;
IF _e52.Q AND NOT CropCut THEN RunSpeed1 := PercentSpeed1; END_IF;
RunSpeedCalculated := _e52.Q;

(* Network 78 *)
WaitToFire1 := Step14 AND LTFires AND ChangeConnector;
WaitCon1 := Step14 AND FeedInitiate;

(* Network 79 *)
TON_10(IN := WaitToFire2, PT := T#50ms);
WaitCon2 := TON_10.Q;

(* Network 80 *)
_e53(CLK := InPosition1);
WaitToFire2 := (_e53.Q OR WaitToFire2) AND NOT WaitCon2;

(* Network 81 *)
WaitCon3 := Step14 AND BeadRollFires AND FeedInitiate;
WaitToFire3 := Step14 AND BeadRollFires;

(* Network 82 *)
_e54(CLK := WaitToFire3);
IF _e54.Q THEN ChangeBeadRoll := TRUE; END_IF;

(* Network 83 *)
Wait1Ready := Step14 AND ((WaitToFire1 AND WaitCon1) OR NOT WaitToFire1);
Wait2Ready := Step14 AND ((WaitToFire2 AND WaitCon2) OR NOT WaitToFire2);
Wait3Ready := Step14 AND ((WaitToFire3 AND WaitCon3) OR NOT WaitToFire3);

(* Network 84 *)
IF (Step15 AND ShearFires) OR (NOT InCycle AND CycleShear) THEN
    shearTime := DINT_TO_TIME(ShearDwell);
END_IF;

(* Network 85 *)
_e55(CLK := LTValve);
_e56(CLK := VValve);
_e57(CLK := LHoleValve);
_e58(CLK := InCycle);
TP_11(IN := (_e55.Q OR _e56.Q OR _e57.Q OR _e58.Q) AND ShearAndDieFires, PT := T#2500ms);
DieDoneTimer := TP_11.Q;

(* Network 86 *)
_e59(CLK := DieDoneTimer);
IF _e59.Q THEN ShearAndDieFires := FALSE; END_IF;

(* Network 87 *)
TP_0(IN := (Step15 AND ShearFires AND NOT ShearAndDieFires) OR (NOT InCycle AND CycleShear), PT := shearTime);
ShearValve := TP_0.Q;

(* Network 88 *)
IF CycleShear THEN CycleShear := FALSE; END_IF;

(* Network 89 *)
IF (Step15 AND LTFires) OR (NOT InCycle AND CycleLTDie) THEN LTTime := DINT_TO_TIME(LTDwell); END_IF;

(* Network 90 *)
TP_1(IN := (Step15 AND LTFires) OR (NOT InCycle AND CycleLTDie), PT := LTTime);
LTValve := TP_1.Q;

(* Network 91 *)
IF CycleLTDie THEN CycleLTDie := FALSE; END_IF;

(* Network 92 *)
IF (Step15 AND VFires) OR (NOT InCycle AND CycleVDie) THEN VTime := DINT_TO_TIME(VDwell); END_IF;

(* Network 93 *)
TP_2(IN := (Step15 AND VFires) OR (NOT InCycle AND CycleVDie), PT := VTime);
VValve := TP_2.Q;

(* Network 94 *)
IF CycleVDie THEN CycleVDie := FALSE; END_IF;

(* Network 95 *)
IF (Step15 AND LeftHoleFires) OR (NOT InCycle AND CycleLDie) THEN
    LeftHoleTime := DINT_TO_TIME(LHoleDwell);
END_IF;

(* Network 96 *)
TP_3(IN := (Step15 AND LeftHoleFires) OR (NOT InCycle AND CycleLDie), PT := LeftHoleTime);
LHoleValve := TP_3.Q;

(* Network 97 *)
IF CycleLDie THEN CycleLDie := FALSE; END_IF;

(* Network 98 *)
IF (Step15 AND CenterHoleFires) OR (NOT InCycle AND CycleCDie) THEN
    CenterHoleTime := DINT_TO_TIME(CHoleDwell);
END_IF;

(* Network 99 *)
TP_4(IN := (Step15 AND CenterHoleFires) OR (NOT InCycle AND CycleCDie), PT := CenterHoleTime);
CHoleValve := TP_4.Q;

(* Network 100 *)
IF (Step15 AND RightHoleFires) OR (NOT InCycle AND CycleRDie) THEN
    RightHoleTime := DINT_TO_TIME(RHoleDwell);
END_IF;

(* Network 101 *)
TP_5(IN := (Step15 AND RightHoleFires) OR (NOT InCycle AND CycleRDie), PT := RightHoleTime);
RHoleValve := TP_5.Q;

(* Network 102 *)
IF (Step15 AND CustomLTFires) OR (NOT InCycle AND CycleCustomLTDie) THEN
    CustomLTTime := DINT_TO_TIME(CustomLTDwell);
END_IF;

(* Network 103 *)
TP_6(IN := (Step15 AND CustomLTFires) OR (NOT InCycle AND CycleCustomLTDie), PT := CustomLTTime);
CustomLTValve := TP_6.Q;

(* Network 104 *)
IF (Step15 AND CustomVFires) OR (NOT InCycle AND CycleCustomVDie) THEN
    CustomVTime := DINT_TO_TIME(CustomVDwell);
END_IF;

(* Network 105 *)
TP_7(IN := (Step15 AND CustomVFires) OR (NOT InCycle AND CycleCustomVDie), PT := CustomVTime);
CustomVValve := TP_7.Q;

(* Network 106 *)
_e60(CLK := ButtonBack7);
_e61(CLK := InCycle);
UnlatchButtons := (Step15 AND _e60.Q) OR _e61.Q;

(* Network 107 *)
_e62(CLK := Step15);
CycleButtons := ((_e62.Q AND ButtonFires) OR CycleButtons) AND NOT UnlatchButtons;

(* Network 108 *)
_e63(CLK := ShearClampUpProx);
_e64(CLK := ProcessorDriveEnable);
IF ((Step15 OR ShearBrakeLatch) AND _e63.Q) OR _e64.Q THEN BrakeLatch := FALSE; END_IF;
UnlatchBender := ((Step15 OR ShearBrakeLatch) AND _e63.Q) OR _e64.Q;

(* Network 109 *)
_e65(CLK := Step15);
CycleMaleBender := ((_e65.Q AND ShearBrakeFires) OR ShearBrakeLatch OR CycleMaleBender) AND NOT UnlatchBender;

(* Network 110 *)
_e66(CLK := Step15);
ChangeKDRolls := _e66.Q AND CleatFires;

(* Network 111 *)
LeftKnockDownRoll := (ChangeKDRolls AND LeftCleatEnable AND NOT LeftKnockDownRoll) OR (LeftKnockDownRoll AND InCycle AND NOT ChangeKDRolls);

(* Network 112 *)
RightKnockDownRoll := (ChangeKDRolls AND RightCleatEnable AND NOT RightKnockDownRoll) OR (RightKnockDownRoll AND InCycle AND NOT ChangeKDRolls);

(* Network 113 *)
ThirdOff1 := NOT ShearValve AND NOT ShearAndDieFires AND NOT LTValve AND NOT VValve AND NOT LHoleValve;

(* Network 114 *)
ThirdOff2 := NOT CHoleValve AND NOT RHoleValve AND NOT ChangeKDRolls AND NOT CycleMaleBender;

(* Network 115 *)
ThirdOff3 := NOT CycleButtons AND NOT CustomLTValve AND NOT CustomVValve AND NOT WaitCon3;

(* Network 116 *)
_e67(CLK := Step17);
IF _e67.Q THEN DieUpTime := DINT_TO_TIME(DieUpDelay); END_IF;

(* Network 117 *)
TON_0(IN := Step17 AND NOT GStep18, PT := DieUpTime);
DieDelayDone := TON_0.Q;

(* Network 118 *)
IncPartsMade := PartCutOff;

(* Network 119 *)
_e68(CLK := GStep18);
IF _e68.Q THEN GTime := DINT_TO_TIME(GapTime); END_IF;

(* Network 120 *)
TP_8(IN := GStep18 AND PartCutOff AND DuctoAuto, PT := GTime);
GapTP := TP_8.Q;

(* Network 121 *)
_e69(CLK := GStep18);
GapPulse := GapTP OR _e69.Q;

(* Network 122 *)
_e70(CLK := GStep18);
IF _e70.Q AND IncPartsMade THEN
    PartsMade := PartsMade + 1;
    RTotalInches := PartLength + RTotalInches;
END_IF;

(* Network 123 *)
IF ChangeJob1 THEN PartsMade := 0; END_IF;

(* Network 124 *)
TotalInches := RTotalInches;

(* Network 125 *)
IF ClearLengthCountSignal THEN RTotalInches := 0; END_IF;
_p71 := ClearLengthCountSignal;
IF _p71 THEN ClearLengthCountSignal := FALSE; END_IF;

(* Network 126: Set StartSignal for touchscreen. Do the warning while waiting for data. Touchscreen resets StartSignal at the tail end of the data transfer. *)
Step01 := (FeedInitiate OR Step01) AND InCycle;

(* Network 127 *)
Step02 := (StartSignal OR Step02) AND Step01;

(* Network 128 *)
Step03 := (WarningComplete OR Step03) AND Step02;

(* Network 129 *)
Step04 := (NOT StartSignal OR Step04) AND Step03;

(* Network 130: Position material for no crop cut. Latch these rungs in if crop cutting. *)
_e72(CLK := MatlAtMeasureRoll);
Step04A := (_e72.Q OR NOT ZeroCropCut OR Step04A) AND Step04;

(* Network 131 *)
Step04B := (ZCReverseComplete OR NOT ZeroCropCut OR Step04B) AND Step04A;

(* Network 132 *)
Step04C := (DirectionDelayDone OR NOT ZeroCropCut OR Step04C) AND Step04B;

(* Network 133 *)
_e73(CLK := MatlAtMeasureRoll);
Step04D := (_e73.Q OR NOT ZeroCropCut OR Step04D) AND Step04C;

(* Network 134 *)
Step04E := (ZCSettleComplete OR Step04E) AND Step04D;

(* Network 135 *)
Step05A := (ServoLoop1Closed OR Step05A) AND Step04E;

(* Network 136 *)
Step05B := (PartRefOK OR Step05B) AND Step05A;

(* Network 137: The last step in the sequence determines if the processor should stop to wait for the FeedInitiate signal. The manual signal is set if the processor needs to stop. The manual signal ujnlatches all steps past Step05B and the waits at Step05B for for FeedInitiate. The auto signal is set if the processor can continue without a FeedInitiate signal. The auto signal unlatches all steps past Step06. *)
_e74(CLK := Step05B);
Step06 := (FeedInitiate OR _e74.Q OR Step06) AND Step05B AND NOT GManualSignal;

(* Network 138 *)
Step07 := (InitMoveSignal OR Step07) AND Step06 AND NOT AutoSignal;

(* Network 139: Step08 enables the the rungs that determine the length of the next move and what to do when it completes. This will execute multiple times in some cases before it is finished. *)
Step08 := (DataUpdated OR Step08) AND Step07 AND NOT NextMoveLookAgain;

(* Network 140 *)
Step08A := (NextMoveDone OR Step08A) AND Step08;

(* Network 141 *)
Step08B := (UpdateTablesDone OR Step08B) AND Step08A;

(* Network 142 *)
Step09 := (NextMoveComplete OR Step09) AND Step08B;

(* Network 143 *)
Step10 := (ClearEncoderSignal OR Step10) AND Step09;

(* Network 144 *)
GStep11 := (RunSpeedCalculated OR GStep11) AND Step10;

(* Network 145 *)
GStep12 := (GFeedMoveQed OR GStep12) AND GStep11;

(* Network 146 *)
Step13 := (NOT InPosition1 OR Step13) AND GStep12;

(* Network 147 *)
Step14 := (InPosition1 OR Step14) AND Step13;

(* Network 148: Dies fire when Step15 latches. Step16 latches when when a die fires or another operation begins. Step17 latches when all operations are finished. *)
Step15 := ((Wait1Ready AND Wait2Ready AND Wait3Ready) OR Step15) AND Step14;

(* Network 149 *)
Step16 := (NOT ThirdOff1 OR NOT ThirdOff2 OR NOT ThirdOff3 OR Step16) AND Step15;

(* Network 150 *)
Step17 := ((ThirdOff1 AND ThirdOff2 AND ThirdOff3) OR Step17) AND Step16;

(* Network 151 *)
GStep18 := (DieDelayDone OR GStep18) AND Step17;

(* Network 152 *)
Step18A := ((GapPulse AND PartCutOff AND DuctoAuto) OR NOT PartCutOff OR NOT DuctoAuto OR Step18A) AND GStep18;

(* Network 153 *)
ShearHitsLTZero := ShearHits < 0;

(* Network 154 *)
GStep18B := (NOT GapPulse OR ShearHitsLTZero OR NOT DuctoAuto OR GStep18B) AND Step18A;

(* Network 155 *)
GStep19 := (NOT ShearFires OR (ShearFires AND ((NOT MakeShearTable AND NOT OneMorePart) OR (NOT DuctoAuto AND OneMorePart))) OR GStep19) AND GStep18B;

(* Network 156 *)
GManualSignal := GStep19 AND NOT ShearHitsLTZero AND ShearFires AND (CropCut OR (PartCutOff AND NOT DuctoAuto));
AutoSignal := GStep19 AND NOT ShearHitsLTZero AND (NOT ShearFires OR (ShearFires AND ((NOT PartCutOff AND NOT CropCut) OR (PartCutOff AND DuctoAuto))));

(* Network 157 *)
Step20 := (ShearHitsLTZero OR Step20) AND GStep19;

(* Network 158 *)
GStep21 := (ReturnCalculated OR GStep21) AND Step20;

(* Network 159 *)
ReturnComplete := ActlMetalEncoder <= ReturnTarget;

(* Network 160 *)
_e75(CLK := MatlAtMeasureRoll);
Step22 := (ReturnComplete OR _e75.Q OR Step22) AND GStep21;

(* Network 161 *)
IF GManualSignal AND ShearFires AND CropCut THEN CropCut := FALSE; END_IF;

(* Network 162 *)
IF NOT InCycle AND NOT CropCut THEN CropCut := TRUE; END_IF;

(* Network 163 *)
IF AutoSignal AND ZeroCropCut THEN ZCOLT0 := ZeroCropOffset <= 0; END_IF;

(* Network 164 *)
_e76(CLK := Step20);
IF _e76.Q THEN
    ReturnTarget := ActlMetalEncoder - REAL_TO_DINT(ZeroCropOffset*UnitsPerInch1*MetalScaler);
END_IF;
ReturnCalculated := _e76.Q;

(* Network 165 *)
IF ZCOLT0 THEN
    CropCut := FALSE;
    ZeroCropCut := FALSE;
END_IF;

(* Network 166 *)
LeftPosA := LeftDiePosition[LeftShuttleIndex];

(* Network 167 *)
_e77(CLK := LHoleValve);
_e78(CLK := InCycle);
IF _e77.Q OR _e78.Q THEN GChangeLShuttle := TRUE; END_IF;

(* Network 168 *)
_e79(CLK := Step09);
GLShuttleUnlatch := GChangeLShuttle AND _e79.Q;
IF GChangeLShuttle AND _e79.Q THEN GChangeLShuttle := FALSE; END_IF;

(* Network 169 *)
LeftShuttleOutput := ((LeftPosA AND GLShuttleUnlatch) OR (LeftShuttleOutput AND NOT GLShuttleUnlatch)) AND InCycle;
END_PROGRAM
```
